(* --> NC-CAM Errors <--*)
		18944	:		FC_NcErrorMsg:='	Nc Cam Errors-	parameter:	"Table ID not allowed" The value for the table ID is not allowed, e.g. because it has already been assigned, is less than or equal to zero, or is greater than 255. 		';
		18945	:		FC_NcErrorMsg:='	Nc Cam Errors-	parameter	:	"Table type not allowed" The value for the table type is unacceptable because it is not defined. 		';
		18946	:		FC_NcErrorMsg:='	Nc Cam Errors-	parameter	:	"Number of lines in the table not allowed" The value of the number of lines in the table is not allowed, because for example, it is smaller than two at linear interpolation and smaller than four at spline interpolation. 		';
		18947	:		FC_NcErrorMsg:='	Nc Cam Errors-	parameter	:	"Number of columns in the table is not allowed" The value of the number of columns in the table is not allowed, because for example, it is less than or equal to zero (depends upon the type of table or slave). 		';
		18948	:		FC_NcErrorMsg:='	Nc Cam Errors-	parameter	:	"JogStep size (position delta) not allowed" The value for the JogStep size between two lines (position delta) is not allowed, because for example, it is less than or equal to zero. 		';
		18949	:		FC_NcErrorMsg:='	Nc Cam Errors-	parameter	:	"Period not allowed" The value for the period is not allowed, because for example, it is less than or equal to zero. 		';
		18950	:		FC_NcErrorMsg:='	Nc Cam Errors-	parameter	:	"Table is not monotonic" The value for the JogStep size is not allowed, because for example, it is less than or equal to zero.		';
		18951	:		FC_NcErrorMsg:='	Nc Cam Errors-	initialization	:	„Table sub type is not allowed” The value for the table sub type is not allowed or otherwise the table class (slave type) do not match up to the table main type.$NTable sub type: (1) equidistant linear position table, (2) equidistant cyclic position table, (3) none equidistant linear position table, (4) none equidistant cyclic position table		';
		18952	:		FC_NcErrorMsg:='	Nc Cam Errors-	initialization	:	„Table interpolation type is not allowed” The value for the table interpolation type is allowed$NTable interpolation type: (0) linear-interpolation, (1) 4-point-interpolation, (2) spline-interpolation		';
		18953	:		FC_NcErrorMsg:='	Nc Cam Errors-	initialization	:	"Incorrect table main type" The table main type is unknown or otherwise the table class (slave type) do not match up to the table main type.$NTable main type: (1) camming table, (2) characteristic table, (3) motion FUNCTION table (MF)		';
		18960	:		FC_NcErrorMsg:='	Nc Cam Errors-	initialization	:	"Table initialisation" Table has not been initialised. Although the table has been created, the rest of the initialisation has not been performed. For instance, the number of lines or columns may be less than or equal to zero.	';
		18961	:		FC_NcErrorMsg:='	Nc Cam Errors-	initialization	:	"Not enough memory" Table could not be created, since there is not enough memory.		';
		18962	:		FC_NcErrorMsg:='	Nc Cam Errors-	function	:	"Function not executed, function not available" The function has not been implemented, or cannot be executed, for the present type of table.		';
		18963	:		FC_NcErrorMsg:='	Nc Cam Errors-	function	:	"Line index not allowed" The start line index or the stop line index to be used for read or write access to the table is not allowed. $NFor instance, the line index may be greater than the total number of lines in the table.		';
		18964	:		FC_NcErrorMsg:='	Nc Cam Errors-	function	:	"Column index not allowed" The start column index or the stop column index to be used for read or write access to the table in not allowed. For instance, the column index may be greater than the total number of columns in the table.		';
		18965	:		FC_NcErrorMsg:='	Nc Cam Errors-	function	:	"Number of lines not allowed" The number of lines to be read from or written to the table is not allowed. $NThe number of lines must be an integer multiple of the number of elements in a line (n * number of columns).		';
		18966	:		FC_NcErrorMsg:='	Nc Cam Errors-	function	:	"Number of columns not allowed" The number of columns to be read from or written to the table is not allowed.$NThe number of columns must be an integer multiple of the number of elements in a column (n * number of lines).  		';
		18967	:		FC_NcErrorMsg:='	Nc Cam Errors-	function	:	"Error in scaling or in range entry" The entries in the table header are inconsistent, e.g. the validity range is empty. $NIf the error is generated during the run time it is a run time error and stops the master/slave group.		';
		18968	:		FC_NcErrorMsg:='	Nc Cam Errors-	function	:	"Multi table slave out of range" The slave master position is outside the table values for the master. The error is a run-time error, and stops the master/slave group.		';
		18969	:		FC_NcErrorMsg:='	Nc Cam Errors-	function	:	"Solo table underflow" The slave master position is outside the table values for the master. The master value of the equidistant table, to be processed linearly, lies under the first table value. $NThe error is a run-time error, and stops the master/slave group.		';
		18970	:		FC_NcErrorMsg:='	Nc Cam Errors-	function	:	"Solo table overflow" The slave master position is outside the table values for the master. The master value of the equidistant table, to be processed linearly, lies above the first table value. $NThe error is a run-time error, and stops the master/slave group.		';
		18971	:		FC_NcErrorMsg:='	Nc Cam Errors-	parameter	:	"Incorrect execution mode" The cyclic execution mode can only be "true" or "false".		';
		18972	:		FC_NcErrorMsg:='	Nc Cam Errors-	parameter	:	"Impermissible parameter" The Fifo parameter is not allowed.		';
		18973	:		FC_NcErrorMsg:='	Nc Cam Errors-	parameter	:	"Fifo is empty" The Fifo of the external generator is empty. This can signify end of track or a run time error.		';
		18974	:		FC_NcErrorMsg:='	Nc Cam Errors-	parameter	:	"Fifo is full" The Fifo of the external generator is full. It is the user‘s task to continue to attempt to fill the Fifo with the rejected values.		';
		18975	:		FC_NcErrorMsg:='	Nc Cam Errors-	parameter	:	„Point-Index of Motion Function invalid”  The point index of a Motion Function Point of a Function Table is invalid. $NFirst the point index has to be larger than zero and second it has to be numerical continuously for one column in the Montion Function Table (e.g. 1,2,3,... or 10,11,12,...).$NnRemark: The point index is not online-changeable but must be constant.		';
		18976	:		FC_NcErrorMsg:='	Nc Cam Errors-	initialization	:	„No diagonalisation of  matrix” The spline can not be calculated. The master positions are not correct.		';
		18977	:		FC_NcErrorMsg:='	Nc Cam Errors-	initialization	:	„Number of spline points to less” The number of points of a cubic spline has to be greater than two.		';
		18978	:		FC_NcErrorMsg:='	Nc Cam Errors-	initialization	:	„Fifo must not be overwritten” Fifo must not be overwritten since then the active line would be overwritten. $NIt is the task of the user to secure that the active line is not modified.		';


(* --> NC-PLC Errors <--*)

		19200	:		FC_NcErrorMsg:='NC-PLC Errors-Parameter:"Axis has been stopped" The axis has been stopped while the axis moves to target position.  The axis could be stopped with a PLC Command via ADS, with the call of AXFNC or with the TwinCAT System Manager.';
		19201	:		FC_NcErrorMsg:='NC-PLC Errors-Parameter:"Axis cannot be started" The axis cannot be started, because: the axis is in an error state, the axis is doing another job,  The axis in protected mode, the axis is not in a ready state.';
		19202	:		FC_NcErrorMsg:='NC-PLC Errors-Parameter:"Control mode not allowed" No Target Position Control and no Position Area Control.';
		19203	:		FC_NcErrorMsg:='NC-PLC Errors-Parameter:"Axis is not moving" Restart position and velocity is only allowed if axis is physically moving.';
		19204	:		FC_NcErrorMsg:='NC-PLC Errors-Parameter:"Wrong mode for RestartPosAndVelo" Wrong mode.';
		19205	:		FC_NcErrorMsg:='NC-PLC Errors-Parameter:"Command not allowed": Endless move to a non specified direction;Read/Write parameter: type mismatch';
		19206	:		FC_NcErrorMsg:='NC-PLC Errors-Parameter:"Parameter not correct"	:Wrong override: > 100% or < 0%	;Wrong gearing factor: RatioDenominator = 0	;Wrong register into process (Register communication)';
		19207	:		FC_NcErrorMsg:='NC-PLC Errors-Parameter:"Timeout axis function block":After positioning, all "MC_Move..." blocks check whether positioning was completed successfully. In the simplest case, the "AxisHasJob" flag of the NC axis is checked, which initially signifies that positioning was logically completed. Depending on the parameterisation of the NC axis,  further checks (quality criteria) are used:"Position range monitoring"	If position range monitoring is active,  the system waits for feedback from the NC.  After positioning, the axis must be within the specified positioning range window. If necessary, the position controller ensures that the axis is moved to the target position.  If the position controller is switched off (Kv=0) or weak, the target may not be reached."Target position monitoring" If target position monitoring is active, the system waits for feedback from the NC.  After positioning, the axis must be within the specified target position window for at least the specified time.  If necessary, the position controller ensures that the axis is moved to the target position.  If the position controller is switched off (Kv=0) or weak, the target may not be reached.  Floating position control may lead to the axis oscillating around the window but not remaining inside the window. If the axis is logically at the target position (logical standstill) but the parameterised position window has not been reached,  monitoring of the above-mentioned NC feedback is aborted with error 19207 (0x4B07) after a constant timeout of 6 seconds. ';
		19208	:		FC_NcErrorMsg:='NC-PLC Errors-Parameter:"Axis in protected mode" Axis is in protected mode (i.e. coupled) and cannot be moved.';
		19209	:		FC_NcErrorMsg:='NC-PLC Errors-Parameter:"Axis is not ready" Axis is not ready and cannot be moved.';
		19210	:		FC_NcErrorMsg:='NC-PLC Errors-Parameter:"Homing error" The Homing of an axis could not be started or was not successful';
		19211	:		FC_NcErrorMsg:='NC-PLC Errors-Parameter:"Invalid definition trigger input definition" The definition of the trigger signal used with the function block MC_TouchProbe is invalid.  The defined encoder ID, the trigger signal or the trigger signal edge are invalid.';
		19212	:		FC_NcErrorMsg:='NC-PLC Errors-Function:"position latch has been deactivated" The function block MC_TouchProbe encountered that a touch probe sequence has been deactivated after the block started this sequence.  The reason for instance can be an axis reset.';
		19213	:		FC_NcErrorMsg:='NC-PLC Errors-Function:"Timeout NC status feedback" A function block has successfully executed a command but the NC does not pass the expected feedback in the axis status word.';
		19214	:		FC_NcErrorMsg:='NC-PLC Errors-Function:"Supplement not installed" - The function is available as supplement product but not installed on the system.';
		19215	:		FC_NcErrorMsg:='NC-PLC Errors-Function:"Timeout Register Access" - The access to a bus terminal register timed out.';
		19216	:		FC_NcErrorMsg:='NC-PLC Errors-Function:"M-Function request missing" This error occurs if a confirmation of an M-Function is made but the request bit is not set.';
		19217	:		FC_NcErrorMsg:='NC-PLC Errors-Parameter:"Zero shift index is out of range" The index of the zero shift is invalid';
		19218	:		FC_NcErrorMsg:='NC-PLC Errors-Parameter:"R parameter index or size is invalid". This error occurs, if the R parameters are written or read and the index or size is out of range';
		19219	:		FC_NcErrorMsg:='NC-PLC Errors-Parameter:"Index for tool description is invalid"';
		19220	:		FC_NcErrorMsg:='NC-PLC Errors-Function:"Version of cyclic channel interface does not match to the requested function and function block, resp."  This error occurs, if an older TwinCAT Version is used and a new functionality from a newer TcNci.lib is called.';
		19221	:		FC_NcErrorMsg:='NC-PLC Errors-Function:"Channel is not ready for requested function". The requested function can not be executed due to a wrong state of the channel.  This error occurs for instance, if retrace is requested and the axes are not stopped with ItpEStop before.';
		19222	:		FC_NcErrorMsg:='NC-PLC Errors-Function:"Requested function is not turned on". The requested function requires an explicit activation before it can be executed.';
		19232	:		FC_NcErrorMsg:='NC-PLC Errors-Parameter:"Cannot append all axes". This error occurs, if you want to append an auxiliary axes to an interpolation group and the function fails.  Probably a prior assignment of an auxiliary axes was skipped.';
		19248	:		FC_NcErrorMsg:='NC-PLC Errors-Parameter:"Pointer invalid". The pointer to a data structure is invalid, e.g. NULL.:data structure MC_CAM_REF is possibly not initialized';
		19249	:		FC_NcErrorMsg:='NC-PLC Errors-Parameter:"Size of memory invalid". The size parameter is invalid:The value of the size parameter is 0 or less than the size of one element of the addressed data structure. The value of the size parameter is less than the requested amount of data. The value of the size parameter does not match other parameters as number of points, number of rows or number of columns.';
		19250	:		FC_NcErrorMsg:='NC-PLC Errors-Parameter:"Invalid cam table ID". The cam table ID is out of the range from 1 to 255.';
		19251	:		FC_NcErrorMsg:='NC-PLC Errors-Parameter:"Invalid point ID". The point ID of a motion function point is lower than 1.';
		19252	:		FC_NcErrorMsg:='NC-PLC Errors-Parameter:"Invalid number of points ". The number of points to read or write is less than 1.';
		19253	:		FC_NcErrorMsg:='NC-PLC Errors-Parameter:"Invalid MC table type". The type of a cam table does not match the MC_TableType definition.';
		19254	:		FC_NcErrorMsg:='NC-PLC Errors-Parameter:"Invalid number of rows". The number of rows of a cam table is less than 1.';
		19255	:		FC_NcErrorMsg:='NC-PLC Errors-Parameter:"Invalid number of columns". The number of columns of a cam table is invalid. The number of columns of a motion function is not equal to 1 ;The number of columns of a standard cam table is not equal to 2 The number of columns does not match other parameters (ValueSelectMask)';
		19256	:		FC_NcErrorMsg:='NC-PLC Errors-Parameter:"Invalid Increment". The increment for an interpolation is invalid, e.g. <= 0.';
		19264	:		FC_NcErrorMsg:='NC-PLC Errors-Monitoring:"Unsupported Terminal Type". The terminal in use is not supported by this function block.';
		19265	:		FC_NcErrorMsg:='NC-PLC Errors-Monitoring:"Register Read/Write Error". This error implies to be a validation error.';
		19266	:		FC_NcErrorMsg:='NC-PLC Errors-Monitoring:"Axis is Enabled". Axis is enabled and is not supposed to be enabled for this operation';
		19267	:		FC_NcErrorMsg:='NC-PLC Errors-Parameter:"Size of compensation table wrong". The stated table size in bytes is not conform with the real size.';
		19268	:		FC_NcErrorMsg:='NC-PLC Errors-Parameter:The minimum/ maximum position of the compenstation table is not conform to the position in the table description (ST_CompensationDesc)';
		19269	:		FC_NcErrorMsg:='NC-PLC Errors-Parameter:"Not implemented". The requested function is not implemented in this combination.';
		19296	:		FC_NcErrorMsg:='NC-PLC Errors-Monitoring:"Motion command not be activated". A motion command has been started and has been buffered and confirmed by the NC. Nevertheless the command did not become active.';
		19297	:		FC_NcErrorMsg:='NC-PLC Errors-Monitoring:"Motion command could not be monitored by the PLC". A motion command has been started and has been buffered and confirmed by the NC.  The PLC has not been able to monitor the execution of this command and the execution status is unclear since the NC is already executing a more recent command.  This error may com up with very short buffered motion commands which are executed during one PLC cycle.';
		19298	:		FC_NcErrorMsg:='NC-PLC Errors-Monitoring:"Buffered command finished with error". A buffered command finished with an error. The error number is not available because a new command is already in execution.';
		19299	:		FC_NcErrorMsg:='NC-PLC Errors-Monitoring:"Buffered command finished without state feedback". A buffered command finished without success or error feedback.';
		19300	:		FC_NcErrorMsg:='NC-PLC Errors-Monitoring:" "BufferMode" not supported". The "BufferMode" is not supported by the command.';
		19301	:		FC_NcErrorMsg:='NC-PLC Errors-Monitoring:"Command number is zero". The system administrated command number for buffered commands is zero.';
		19313	:		FC_NcErrorMsg:='NC-PLC Errors-Parameter:"Invalid NCI Entry Type". FB_NciFeedTablePreparation is called with an unknown nEntryType';
		19314	:		FC_NcErrorMsg:='NC-PLC Errors-Function:"NciFeedTable full". The table is full filled and therefore this entry is not accepted. To do:Transfer the context of the table with FB_NciFeedTable to the NC-Kernel.  If this succeeded bFeedingDone becomes TRUE and the context of the table has to be reset with bResetTable (FB_NciFeedTablePreparation).  Now the table can be refilled with new entries.';
		19315	:		FC_NcErrorMsg:='NC-PLC Errors-Function:internal error';
		19316	:		FC_NcErrorMsg:='NC-PLC Errors-Parameter:$NST_NciTangentialFollowingDesc: tangential axis is not an auxiliary axis"  The entry ST_NciTangentialFollowingDesc contains an tangential axis that is no auxiliary axis.';
		19317	:		FC_NcErrorMsg:='NC-PLC Errors-Parameter:$NST_NciTangentialFollowingDesc: nPathAxis1 and nPathAxis2, resp. are no path axes. So it is not possible to determine the plane.';
		19318	:		FC_NcErrorMsg:='NC-PLC Errors-Parameter:$NST_NciTangentialFollwoingDesc: nPathAxis1 and nPathAxis2 are equal. So it is not possible to determine the plane.';
		19319	:		FC_NcErrorMsg:='NC-PLC Errors-Parameter:$NST_NciGeoCirclePlane: circle is programmed in a wrong manner.';
		19320	:		FC_NcErrorMsg:='NC-PLC Errors-Function:$NInternal error in calculation of the tangential following';
		19321	:		FC_NcErrorMsg:='NC-PLC Errors-Monitoring:$NTangential following: With ST_NciTangentialFollowingDesc the monitoring of the deviation angle (E_TfErrorOnCrirical1)  is activated and with the actual segment the deviation angle is too big.';
		19322	:		FC_NcErrorMsg:='NC-PLC Errors-Function:$Nnot implemented';
		19323	:		FC_NcErrorMsg:='NC-PLC Errors-Parameter:$NTangential Following: The radius of the actual circle segment is too small';
		19324	:		FC_NcErrorMsg:='NC-PLC Errors-Parameter:$NFB_NciFeedTablePreparation: pEntry is NULL';
		19325	:		FC_NcErrorMsg:='NC-PLC Errors-Parameter:$NFB_NciFeedTablePreparation: The specified nEntryType does not match the the structure type';
		19326	:		FC_NcErrorMsg:='NC-PLC Errors-Parameter:$NST_NciMFuncFast and ST_NciMFuncHsk: The requested m-function is not in between 0..159';
		19327	:		FC_NcErrorMsg:='NC-PLC Errors-Parameter:$NST_NciDynOvr: The requested value for the dynamic override is not in between 0.01 and 1.0';
		19328	:		FC_NcErrorMsg:='NC-PLC Errors-Parameter:$NST_NciVertexSmoothing: invalid parameter. This error occurs with a negative vertex radius or an unknown vertex smoothing type.';
		19329	:		FC_NcErrorMsg:='NC-PLC Errors-Parameter:$NFB_NciFeedTablePrepartion: The requested velocity is not in a valid range';
		19330	:		FC_NcErrorMsg:='NC-PLC Errors-Parameter:$NST_Nci*: invalid parameter';



		33056	:	FC_NcErrorMsg:='NC3_Environment_Invalid configuration for Object (e.g. in System Manager)';
		33057	:	FC_NcErrorMsg:='NC3_Environment_Invalid environment FOR Object (e.g. TcCom-Object Hierarchy OR missing/faulty Objects)';
		33058	:	FC_NcErrorMsg:='NC3_Environment_Incompatible Driver OR Object';
		33084	:	FC_NcErrorMsg:='NC3_Parameter_BufferMode is invalid';
		33085	:	FC_NcErrorMsg:='NC3_FunctionBlock_Only one active Instance OF FUNCTION Block per Group is allowed';
		33086	:	FC_NcErrorMsg:='NC3_State_Command is NOT allowed in current group state';
		33087	:	FC_NcErrorMsg:='NC3_FunctionBlock_Slave cannot synchronize.The slave cannot reach the SlaveSyncPosition BY the TIME the master has reached the MasterSyncPos';
		33088	:	FC_NcErrorMsg:='NC3_Parameter_Invalid value FOR one OR more OF the dynamic parameters (A, D, J)';
		33089	:	FC_NcErrorMsg:='NC3_Parameter_IdentInGroup is invalid';
		33090	:	FC_NcErrorMsg:='NC3_Parameter_The number OF axes in the group is incompatible with the axes convention';
		33091	:	FC_NcErrorMsg:='NC3_Communication_FUNCTION Block OR respective Command is NOT supported BY Target';
		33093	:	FC_NcErrorMsg:='NC3_FunctionBlock_Mapping OF Cyclic INTERFACE between Nc AND Plc missing (e.g. AXIS_REF, AXES_GROUP_REF, ...)';
		33094	:	FC_NcErrorMsg:='NC3_FunctionBlock_Invalid Velocity ValueThe velocity was NOT set OR the entered value is invalid';
		33096	:	FC_NcErrorMsg:='NC3_FunctionBlock_Invalid Input Value';
		33097	:	FC_NcErrorMsg:='NC3_FunctionBlock_Invalid OR Incomplete Input ARRAY';
		33098	:	FC_NcErrorMsg:='NC3_Parameter_Unsupported Dynamics FOR selected Group Kernel';
			
		
		ELSE
			IF 36844<error AND error< 36857 THEN
				FC_NcErrorMsg:='NC3_Internal_Unexpected INTERNAL Error';
			ELSE		
				FC_NcErrorMsg:='Msg Unknown';
			END_IF	
END_CASE

END_FUNCTION

// ---- POUs/Lib/Motion/CreateNCErrMsgDetails.TcPOU
FUNCTION CreateNCErrMsgDetails : enumMotorEvents
VAR_INPUT
	Error: UDINT;
END_VAR
VAR
END_VAR

CASE Error OF
		0		: 		
(* --> General NC Errors <--*)
			CreateNCErrMsgDetails := enumMotorEvents.NoEvents;
		16384,16385,16386,16400,16401,16402,16403,16404,16405,16406	:	
			CreateNCErrMsgDetails := enumMotorEvents.MotorGeneralError;
		16416,16417,16418,16419,16420,16421	:
			CreateNCErrMsgDetails := enumMotorEvents.MotorFeedBackErr;
		16432,16433,16448:	
			CreateNCErrMsgDetails := enumMotorEvents.MotorGeneralError;
		16464	,	16465	,16466	:	
			CreateNCErrMsgDetails := enumMotorEvents.MotorFeedBackErr;
		16480,16481	,16482	,16483	,16496	,16497	:		
            CreateNCErrMsgDetails := enumMotorEvents.MotorGeneralError;      
                        
(* --> Channel Errors <-*)
		16641	,	
		16642	,	
		16643	,	
		16644	,	
		16645	,	
		16646	,	
		16647	,	
		16648	,	
		16649	,	
		16650	,	
		16656	,	
		16657	,	
		16658	,	
		16659	,	
		16660	,	
		16661	,	
		16662	,	
		16663	,	
		16672	,
		16673	,	
		16674	,	
		16688	,	
		16689	,	
		16690	,	
		16691	,	
		16704	,	
		16705	,	
		16706	,	
		16707	,	
		16708	,	
		16709	,	
		16720	,	
		16721	,	
		16722	,	
		16723	,	
		16724	,	
		16725	,
		16726	,	
		16727	,	
		16728	,	
		16729	,	
		16730	,	
		16731	,	
		16732	,	
		16733	,	
		16734	,
		16735	,
		16736	,	
		16737	,	
		16738	,	
		16752	,	
		16753	,	
		16754	:	
 			CreateNCErrMsgDetails := enumMotorEvents.MotorGeneralError; 
(* --> Group Errors <--*)

		16896	,	
		16897	,	
		16898	,	
		16899	,	
		16900	,	
		16901	,	
		16902	,	
		16903	,	
		16904	,	
		16905	,	
		16906	,	
		16907	,	
		16908	,	
		16909	,	
		16910	,	
		16911	,	
		16912	,	
		16913	,	
		16914	,	
		16915	,	
		16916	,	
		16917	,	
		16918	,	
		16919	,	
		16920	,	
		16921	,	
		16922	,	
		16923	,	
		16924	,	
		16925	,	
		16926	,	
		16927	,	
		16928	,	
		16929	,	
		16930	:
				CreateNCErrMsgDetails := enumMotorEvents.PLCIllegalParam; 
		16931	:
				CreateNCErrMsgDetails := enumMotorEvents.DriveNotEnabled; 	
		16932	:
				CreateNCErrMsgDetails := enumMotorEvents.MotorGeneralError ;
		16933	:
				CreateNCErrMsgDetails := enumMotorEvents.DriveNotReady ;	
		16934	,	
		16935	:	;
				
		16936	,	
		16937	:	;
				CreateNCErrMsgDetails := enumMotorEvents.MotorGeneralError;	
		16938	:
				CreateNCErrMsgDetails := enumMotorEvents.DriveNotEnabled; 		
		16939	,	
		16940	,	
		16941	,	
		16942	,	
		16943	,	
		16944	,	
		16945	,	
		16946	,	
		16947	,	
		16948	:	;
		16949	,	
		16950	,	
		16951	,	
		16952	,	
		16953	,	
		16954	,	
		16955	,	
		16956	,	
		16957	:	;
		16958	,	
		16959	,	
		16960	,	
		16961	,	
		16962	,	
		16963	,	
		16964	,	
		16965	,	
		16966	:	;
		16967	,	
		16968	,	
		16969	,	
		16970	,	
		16971	,	
		16972	,	
		16973	,	
		16974	,	
		16975	:	;
		16976	,	
		16977	,	
		16978	,	
		16979	:
				CreateNCErrMsgDetails := enumMotorEvents.MotorGeneralError;		
		16980	:
				CreateNCErrMsgDetails := enumMotorEvents.MotorFeedBackErr;			
		16981	,	
		16982	,	
		16983	,	
		16984	:	;
		16985	,	
		16986	,	
		16987	,	
		16988	,	
		16989	,	
		16990	,	
		16991	:
		 		CreateNCErrMsgDetails := enumMotorEvents.MotorGeneralError;	
		16992	:	
				CreateNCErrMsgDetails := enumMotorEvents.DriveNotEnabled ;
		16993	,	
		16994	,	
		16995	,	
		16996	,	
		16997	,	
		16998	,	
		16999	,	
		17000	,	
		17001	,	
		17002	,	
		17003	,	
		17004	,	
		17005	,	
		17006	,	
		17007	,	
		17008	,	
		17009	,	
		17010	,	
		17011	,	
		17012	,	
		17014	,	
		17015	,	
		17017	,	
		17018	,	
		17019	,	
		17020	,	
		17021	,	
		17022	,	
		17023	,	
		17024	,	
		17025	,	
		17026	,	
		17027	,	
		17028	,	
		17029	,	
		17030	,	
		17031	,	
		17032	,	
		17033	,	
		17034	,	
		17035	,	
		17036	,	
		17037	,
		17038	,
		17039	,
		17040	,
		17041	,
		17042	,
		17043	,
		17044	,
		17045	,
		17046	,
		17047	,
		17052	,
		17053	,
		17054	,
		17056	,	
		17057	,	
		17058	,	
		17059	,	
		17060	,	
		17061	,	
		17062	,	
		17063	,	
		17064	,	
		17065	,	
		17066	,	
		17067	,	
		17068	,	
		17069	,	
		17070	,	
		17071	,	
		17072	,	
		17073	,	
		17074	,	
		17075	,	
		17076	,	
		17077	,	
		17078	,	
		17079	,	
		17080	,	
		17082	,	
		17083	,	
		17084	,	
		17085	,	
		17086	,		
		17087	,		
		17088	,		
		17089	,		
		17090	,		
		17091	,		
		17092	,		
		17093	,		
		17094	,		
		17095	,		
		17096	,		
		17097	,		
		17098	,		
		17099	,		
		17100	,		
		17101	,		
		17102	,		
		17103	,		
		17104	,		
		17105	,		
		17106	,		
		17107	,		
		17108	,		
		17109	,		
		17110	,		
		17111	,		
		17112	,		
		17114	,		
		17115	,		
		17116	,		
		17117	,		
		17118	,		
		17119	,		
		17120	,		
		17121	,		
		17122	,		
		17123	,		
		17124	,		
		17125	,		
		17127	,		
		17128	,		
		17129	,		
		17130	,		
		17131	,		
		17132	,		
		17133	,		
		17134	,		
		17135	,		
		17136	,		
		17137	,		
		17138	,		
		17139	,		
		17140	,		
		17142	,		
		17151	:		
               CreateNCErrMsgDetails := enumMotorEvents.MotorGeneralError;	         

(* --> Axis Errors <--*)

		17152	,		
		17153	,		
		17158	,		
		17159	,		
		17160	,		
		17161	,		
		17162	,		
		17163	,		
		17164	,		
		17165	,		
		17166	,		
		17167	,		
		17168	,		
		17170	,		
		17171	,		
		17172	,		
		17173	,		
		17174	,		
		17175	,		
		17176	,		
		17177	,		
		17178	,		
		17179	,		
		17180	,		
		17181	,		
		17182	,		
		17183	,		
		17184	,		
		17185	,		
		17186	,		
		17187	,		
		17188	,		
		17189	,		
		17190	,		
		17191	,		
		17192	,		
		17193	,		
		17194	,		
		17195	,		
		17196	,		
		17197	,		
		17198	,		
		17199	,		
		17200	,		
		17201	,		
		17202	,		
		17203	,		
		17204	,		
		17210	,		
		17211	:	
				CreateNCErrMsgDetails := enumMotorEvents.MotorGeneralError;		
		17216	:		
				CreateNCErrMsgDetails := enumMotorEvents.DriveNotReady ;
		17217	,		
		17218	,		
		17219	,		
		17220	,		
		17221	,		
		17222	,		
		17223	,		
		17224	:
			CreateNCErrMsgDetails := enumMotorEvents.MotorGeneralError;				
		17238	,		
		17239	,		
		17240	:
			CreateNCErrMsgDetails := enumMotorEvents.DriveNotEnabled;
		17241	,		
		17242	,		
		17243	,		
		17244	:
				CreateNCErrMsgDetails := enumMotorEvents.MotorGeneralError;		
		17245	:
				CreateNCErrMsgDetails := enumMotorEvents.MotorPositionError;		
		17246	,		
		17249	,		
		17250	,		
		17251	,		
		17312	:		
	             CreateNCErrMsgDetails := enumMotorEvents.MotorGeneralError;
                        
(* --> Encoder Errors <--*)           
		17408	,		
		17409	,		
		17410	,		
		17411	,		
		17412	,		
		17413	,		
		17414	,		
		17415	,		
		17416	,		
		17417	,		
		17418	,		
		17419	,		
		17420	,		
		17421	,		
		17422	,		
		17423	,		
		17424	,		
		17425	,		
		17426	,		
		17427	,		
		17428	,		
		17429	,		
		17430	,		
		17431	,		
		17432	,		
		17433	,		
		17434	,		
		17435	,		
		17436	,		
		17440	,		
		17441	,		
		17442	,		
		17443	,		
		17444	,		
		17445	,		
		17446	,		
		17456	,		
		17457	,		
		17458	,		
		17459	,		
		17460	,		
		17461	:		
		        CreateNCErrMsgDetails := enumMotorEvents.MotorGeneralError;
		17472	:
				CreateNCErrMsgDetails := enumMotorEvents.DriveNotReady;		
		17473	,	
		17474	,		
		17475	:
  				CreateNCErrMsgDetails := enumMotorEvents.MotorGeneralError;		
		17488	,  				
		17489	:
				CreateNCErrMsgDetails := enumMotorEvents.MotorFeedBackErr;				
		17504	,		
		17505	,		
		17506	,		
		17507	:
				CreateNCErrMsgDetails := enumMotorEvents.MotorGeneralError;				
		17508	,		
		17509	:
				CreateNCErrMsgDetails := enumMotorEvents.MotorFeedBackErr;
			
		17510   :
				CreateNCErrMsgDetails := enumMotorEvents.DriveComError;
	 
		17520	,	
		17570	,	
		17571	:
			CreateNCErrMsgDetails := enumMotorEvents.MotorGeneralError;	

(* --> Controller Errors <--*)
		17664	,
		17665	, 
		17666	,
		17667	,
		17668	,
		17669	,
		17670	,
		17671	,
		17672	,
		17673	,
		17680	,
		17681	,
		17682	,
		17683	,
		17684	,
		17685	,
		17686	,
		17687	,
		17688	,
		17689	,
		17690	,
		17691	,
		17692	,
		17693	,
		17696	,
		17697	,
		17698	,
		17699	,
		17700	:
			CreateNCErrMsgDetails := enumMotorEvents.MotorGeneralError;	
		17728	:
			CreateNCErrMsgDetails := enumMotorEvents.DriveNotReady;
		17729	,	
		17730	:
			CreateNCErrMsgDetails := enumMotorEvents.MotorGeneralError;		
		17744	:
			CreateNCErrMsgDetails := enumMotorEvents.MotorPositionError;
		17745	:
			CreateNCErrMsgDetails := enumMotorEvents.MotorSpeedError;
		17824	,	
		17825	,	
		17826	,	
		17827	,	
		17828	:	
			CreateNCErrMsgDetails := enumMotorEvents.MotorGeneralError;	

(* --> Drive Errors <--*)

		17920	,
		17921	,
		17922	,
		17923	,
		17924	,
		17925	,
		17926	,
		17927	,
		17928	,
		17929	,
		17930	, 
		17931	,
		17932	,
		17933	,
		17935	,
		17936	,
		17937	,	
		17938	,
		17939	,
		17940	,
		17941	,
		17942	,
		17943	,
		17952	,
		17953	,
		17954	,
		17955	,
		17956	,
		17959	:
			CreateNCErrMsgDetails := enumMotorEvents.MotorGeneralError;	

		17968	:
			CreateNCErrMsgDetails := enumMotorEvents.MotorOverTemp;	
		17969	,
		17970	,
		17971	:
			CreateNCErrMsgDetails := enumMotorEvents.MotorSupplyError;
		17972	,
		17973	:
			CreateNCErrMsgDetails := enumMotorEvents.MotorOverCurrent;
		17974	:
			CreateNCErrMsgDetails := enumMotorEvents.MotorStalled;
		17984	:
			CreateNCErrMsgDetails := enumMotorEvents.DriveNotReady;
		17985	,
		17986	,
		17987	:
			CreateNCErrMsgDetails := enumMotorEvents.MotorGeneralError;	
		18000	:
			CreateNCErrMsgDetails := enumMotorEvents.DriveNotReady;	
		18001	:
			CreateNCErrMsgDetails := enumMotorEvents.DriveComError;
		18002	:
			CreateNCErrMsgDetails := enumMotorEvents.MotorGeneralError;	
		18005	:
			CreateNCErrMsgDetails := enumMotorEvents.DriveComError;

(* --> NC-CAM Errors <--*)
		18944	, 
		18945	, 
		18946	, 
		18947	, 
		18948	, 
		18949	, 
		18950	, 
		18951	, 
		18952	, 
		18953	, 
		18960	, 
		18961	, 	
		18962	, 	
		18963	, 
		18964	, 
		18965	, 
		18966	,	
		18967	, 
		18968	, 	
		18969	, 
		18970	, 
		18971	, 	
		18972	,	
		18973	,	
		18974	,	
		18975	,
		18976	,	
		18977	,	
		18978	,	
		18979   : 
			CreateNCErrMsgDetails := enumMotorEvents.MotorGeneralError;
(* --> NC-PLC Errors <--*)

		19200	,	
		19201	,	
		19202	,	
		19203	,	
		19204	,	
		19205	,	
		19206	,	
		19207	,
		19208	,	
		19209	,	
		19210	,	
		19211	,	
		19212	,	
		19213	,	
		19214	,	
		19215	,	
		19216	,	
		19217	,
		19218	,
		19219	,
		19220	,
		19221	,
		19222	,
		19232	,
		19248	:	;
		19249	,
		19250	,
		19251	,
		19252	,
		19253	,
		19254	,
		19255	,
		19256	,
		19264	,
		19265	,
		19266	,
		19267	,
		19268	,
		19269	,
		19296	,
		19297	,
		19298	,
		19299	,
		19300	,
		19301	,
		19313	,
		19314	,
		19315	,
		19316	,
		19317	,
		19318	,
		19319	,
		19320	,
		19321	,
		19322	,
		19323	,
		19324	,
		19325	,
		19326	,
		19327	,
		19328	,
		19329	,
		19330	,
		19344   ,
		19345   ,
		19346   ,
		19347   ,
		19348   ,
		19349   ,
		19350   ,
		19351   ,
		19352   ,
		19360   ,
		19361   ,
		19376   ,
		19377   ,
		19378   ,
		19379   ,
		19380   ,
		19381   :
                
            	CreateNCErrMsgDetails := enumMotorEvents.MotorGeneralError;    
		        
                
                
		33056	,
		33057	,
		33058	,
		33084	,
		33085	,
		33086	,
		33087	,
		33088	,
		33089	,
		33090	,
		33091	,
		33093	,
		33094	,
		33096	,
		33097	,
		33098	:	
				CreateNCErrMsgDetails := enumMotorEvents.MotorGeneralError;
		
		ELSE
			IF 36844<error AND error< 36857 THEN
			//
			ELSE		
				//
				CreateNCErrMsgDetails := enumMotorEvents.MotorGeneralError;
			END_IF	
END_CASE

END_FUNCTION

// ---- POUs/Lib/Motion/MultiAxis_FB.TcPOU
FUNCTION_BLOCK PUBLIC MultiAxis_FB
VAR_INPUT
	
	BasicAxisCtrlPtr 	: POINTER TO Basic_axis_typ ;
	MultiAxisCtrlPtr 	: POINTER TO MultiAxis_typ ;
	
END_VAR
VAR_IN_OUT
	MasterRef	:	AXIS_REF;
    MasterRef2 	: 	AXIS_REF;
    MasterRef3 	: 	AXIS_REF;
    MasterRef4 	: 	AXIS_REF;
	AxisRef		: 	AXIS_REF;
END_VAR
VAR_OUTPUT
END_VAR
	
VAR
	LogMsgInit		: BOOL;
	LogMsg_0 		: LogMsg ;
	DecoupleTriger	: Trigger ;
	Decouple		: bool ;
	fbMC_CamTableSelect	: MC_CamTableSelect;
	fbMC_CamIn			: MC_CamIn;
	fbMC_CamOut			: MC_CamOut;
	fbMC_GearInDyn		: MC_GearInDyn;
	fbMC_GearInPos		: MC_GearInPos;
	fbMC_GearOut		: MC_GearOut ;
	fbMC_GearInMultiMaster : MC_GearInMultiMaster ;
	
	ErrorTrig : Trigger ;
	AxisStep : eMultiAxisState ;
	tempTrig : Trigger ;
	
	
	
	tmp_ErrorEntry			: Eh_ErrorEntry_typ;
	
END_VAR

IF NOT LogMsgInit THEN 
	LogMsg_0.logData.category:=	BasicAxisCtrlPtr^.Input.Parameter.ThreadName;     
	LogMsg_0.Enable:= 	TRUE; 	
END_IF

LogMsg_0.ptrGlobalArray:= 	ADR(LogGlobalArray);
LogMsg_0.ptrEncoderAngle:= 	ADR(BasicAxisCtrlPtr^.Input.Parameter.PosForLog);

IF BasicAxisCtrlPtr^.Output.Status.FAULT THEN
	

	AxisStep := MultiAxis_STATE_ERROR;
		
END_IF

//in case of Stop go to CAM_STATE_WAIT
IF (BasicAxisCtrlPtr^.Input.Command.Stop = TRUE) OR (BasicAxisCtrlPtr^.Input.Command.Halt = TRUE) THEN
	AxisStep := MultiAxis_STATE_WAIT;
END_IF

CASE AxisStep OF
		
	(******************** WAIT *************************)
	MultiAxis_STATE_WAIT:  (* STATE: Wait *)
		
		IF BasicAxisCtrlPtr^.Output.Status.ReadyForCmd THEN
			Disable_All_FB(FALSE);
			AxisStep := MultiAxis_STATE_ENTER_READY ;
		END_IF
		
	MultiAxis_STATE_ENTER_READY:
			IF Disable_All_FB(TRUE) THEN
				AxisStep := MultiAxis_STATE_READY ;
			END_IF	

	(******************** READY *************************)
	MultiAxis_STATE_READY:
	
		IF MultiAxisCtrlPtr^.Input.Command.CamTableSelect.Start THEN
			
			MultiAxisCtrlPtr^.Input.Command.CamTableSelect.Start := FALSE ;
			MultiAxisCtrlPtr^.Output.Status.CamTableSelect.Done := FALSE ;
			AxisStep := MultiAxis_STATE_CAM_SELECT ;
			
		ELSIF MultiAxisCtrlPtr^.Input.Command.CamIn.StartSlave THEN
			
			MultiAxisCtrlPtr^.Input.Command.CamIn.StartSlave := FALSE ;
			fbMC_CamIn.Execute := FALSE;	
			AxisStep := MultiAxis_STATE_CAM_START ;
			
		ELSIF MultiAxisCtrlPtr^.Input.Command.CamIn.DisengageSlave THEN
			
			MultiAxisCtrlPtr^.Input.Command.CamIn.DisengageSlave := FALSE ;
			MultiAxisCtrlPtr^.Output.Status.CamOut.Done := FALSE ;
			fbMC_CamOut.Execute := FALSE ;
			AxisStep := MultiAxis_STATE_CAM_STOP ;
			
		ELSIF MultiAxisCtrlPtr^.Input.Command.GearInPos.StartSlave  THEN
			MultiAxisCtrlPtr^.Input.Command.GearInPos.StartSlave := FALSE ;
			MultiAxisCtrlPtr^.Output.Status.GearInPos.InSync := FALSE ;
			MultiAxisCtrlPtr^.Output.Status.GearOut.Done 	:= FALSE ;
			AxisStep := MultiAxis_STATE_GEAR_IN_POS ;
			
		ELSIF MultiAxisCtrlPtr^.Input.Command.GearInDyn.StartSlave THEN
			MultiAxisCtrlPtr^.Input.Command.GearInDyn.StartSlave := FALSE ;
			MultiAxisCtrlPtr^.Output.Status.GearInDyn.InGear := FALSE ;
			MultiAxisCtrlPtr^.Output.Status.GearOut.Done 	:= FALSE ;
			AxisStep := MultiAxis_STATE_GEAR_IN_DYN ;
			
		ELSIF MultiAxisCtrlPtr^.Input.Command.GearInDyn.DisengageSlave THEN
			MultiAxisCtrlPtr^.Input.Command.GearInDyn.DisengageSlave := FALSE ;
			MultiAxisCtrlPtr^.Output.Status.GearInDyn.InGear := FALSE ;
			MultiAxisCtrlPtr^.Output.Status.GearOut.Done 	:= FALSE ;
			MultiAxisCtrlPtr^.Output.Status.GearInMultiMaster.InGear := FALSE ;
			AxisStep := MultiAxis_STATE_GEAR_OUT ;
			
		ELSIF MultiAxisCtrlPtr^.Input.Command.GearInMultiMaster.StartSlave THEN
			MultiAxisCtrlPtr^.Input.Command.GearInMultiMaster.StartSlave := FALSE ;
			MultiAxisCtrlPtr^.Output.Status.GearInMultiMaster.InGear := FALSE ;
			MultiAxisCtrlPtr^.Output.Status.GearOut.Done 	:= FALSE ;
			AxisStep := MultiAxis_STATE_GEAR_IN_MULTI_MASTER;
			
		ELSIF MultiAxisCtrlPtr^.Input.Command.GearInMultiMaster.DisengageSlave THEN
			MultiAxisCtrlPtr^.Input.Command.GearInMultiMaster.DisengageSlave := FALSE ;
			MultiAxisCtrlPtr^.Output.Status.GearInDyn.InGear := FALSE ;
			MultiAxisCtrlPtr^.Output.Status.GearOut.Done 	:= FALSE ;
			MultiAxisCtrlPtr^.Output.Status.GearInMultiMaster.InGear := FALSE ;
			AxisStep := MultiAxis_STATE_GEAR_OUT ;
		END_IF
	
	(******************** CamTableSelect *************************)	
	MultiAxis_STATE_CAM_SELECT:

		IF THIS^.CamTableSelect()THEN
			AxisStep := MultiAxis_STATE_READY;
		END_IF
		
	(******************** START CAM MOVEMENT **********************)	
	MultiAxis_STATE_CAM_START:
	
		fbMC_CamIn.MasterOffset 	:= MultiAxisCtrlPtr^.Input.Parameter.CamIn.MasterOffset;
		fbMC_CamIn.SlaveOffset 		:= MultiAxisCtrlPtr^.Input.Parameter.CamIn.SlaveOffset; 
		fbMC_CamIn.MasterScaling	:= MultiAxisCtrlPtr^.Input.Parameter.CamIn.MasterScaling;
		fbMC_CamIn.SlaveScaling 	:= MultiAxisCtrlPtr^.Input.Parameter.CamIn.SlaveScaling;
		fbMC_CamIn.StartMode 		:= MultiAxisCtrlPtr^.Input.Parameter.CamIn.StartMode;
		fbMC_CamIn.CamTableID 		:= MultiAxisCtrlPtr^.Input.Parameter.CamIn.CamTableID;
		fbMC_CamIn.BufferMode 		:= MultiAxisCtrlPtr^.Input.Parameter.CamIn.BufferMode;
		fbMC_CamIn.Options 			:= MultiAxisCtrlPtr^.Input.Parameter.CamIn.Options; 
		
		fbMC_CamIn.Execute := TRUE;
		AxisStep := MultiAxis_STATE_READY;
		
	(******************** STOP CAM MOVEMENT **********************)
	MultiAxis_STATE_CAM_STOP: (* STATE: Stop electronic gear coupling *)
		
		IF THIS^.CamOut()THEN
			fbMC_CamIn.Execute := FALSE;
			AxisStep := MultiAxis_STATE_READY;
		END_IF	
			
	(******************** GEAR IN DYNAMIC **********************)	
	MultiAxis_STATE_GEAR_IN_DYN:
	
	
		IF (MultiAxisCtrlPtr^.Input.Command.GearInDyn.DisengageSlave)			 
				AND NOT THIS^.GearInDyn() THEN
			AxisStep := MultiAxis_STATE_GEAR_OUT;
		END_IF
				
	(******************** GEAR IN POSITION **********************)
	MultiAxis_STATE_GEAR_IN_POS:
	
		IF MultiAxisCtrlPtr^.Input.Command.GearInPos.DisengageSlave AND NOT THIS^.GearInPos() THEN
			AxisStep := MultiAxis_STATE_GEAR_OUT;
		END_IF
		
		//THIS^.GearInPos();

	(******************** GEAR IN MultiMaster **********************)
	MultiAxis_STATE_GEAR_IN_MULTI_MASTER:
(*	
		IF ((MultiAxisCtrlPtr^.Input.Command.GearInMultiMaster.DisengageSlave) OR (BasicAxisCtrlPtr^.Input.Command.Power = FALSE))  
			AND NOT THIS^.GearInMultiMaster() THEN
				AxisStep := MultiAxis_STATE_GEAR_OUT;
		END_IF
*)

		IF NOT THIS^.GearInMultiMaster() THEN
				AxisStep := MultiAxis_STATE_GEAR_OUT;
		END_IF
			
	(******************** GEAR OUT **********************)	
	MultiAxis_STATE_GEAR_OUT:
		
		IF THIS^.GearOut()THEN
			MultiAxisCtrlPtr^.Output.Status.GearInPos.InSync := FALSE ;
			MultiAxisCtrlPtr^.Output.Status.GearInDyn.InGear := FALSE ;
			MultiAxisCtrlPtr^.Output.Status.GearInMultiMaster.InGear := FALSE ;
			AxisStep := MultiAxis_STATE_READY;
		END_IF
		
	(******************** Error **********************)	
	MultiAxis_STATE_ERROR:	
		
			THIS^.ResetAll_MC_FB();	
		
			IF BasicAxisCtrlPtr^.Output.Status.FAULT THEN						
				AxisStep := MultiAxis_STATE_ERROR;
			ELSE
				MultiAxisCtrlPtr^.Output.Error.ErrorID := 0 ;
				AxisStep := MultiAxis_STATE_WAIT;
			END_IF			
	
	
END_CASE 


IF DecoupleTriger.EDGEPOS(BasicAxisCtrlPtr^.Output.Status.AxisStatus.Error)THEN
	Decouple := TRUE ;
END_IF
IF Decouple THEN	
	IF THIS^.GearOut() THEN
		Decouple := FALSE ;
	END_IF
END_IF

(********************** MC_CAMIN FB Call *************************)
	
THIS^.CamIn();
	
//=====================================================================================================================\\

//IF MultiAxisCtrlPtr^.Output.Error.ErrorID <> 0 THEN
//	BasicAxisCtrlPtr^.Output.Error.ErrorID := MultiAxisCtrlPtr^.Output.Error.ErrorID ;
//	MultiAxisCtrlPtr^.Output.Error.ErrorID := 0;
//END_IF

//fnLogTransfer FUNCTION call
fnLogTransfer(ADR(LogMsg_0));

METHOD AddNCError : BOOL
VAR_INPUT
	ErrorId			: UDINT;
	ErrorPrefix     : STRING[100];
END_VAR

	tmp_ErrorEntry.ErrorId		:= ErrorId;

	tmp_ErrorEntry.ErrorText	:= ErrorPrefix;

	tmp_ErrorEntry.ErrorText	:= CONCAT(tmp_ErrorEntry.ErrorText, UDINT_TO_STRING(tmp_ErrorEntry.ErrorId));
	tmp_ErrorEntry.ErrorText	:= CONCAT(tmp_ErrorEntry.ErrorText, 'Task: ');
	tmp_ErrorEntry.ErrorText	:= CONCAT(tmp_ErrorEntry.ErrorText, MultiAxisCtrlPtr^.Input.Parameter.ThreadName);	
	tmp_ErrorEntry.ErrorText	:= CONCAT(tmp_ErrorEntry.ErrorText, FC_NcErrorMsg(tmp_ErrorEntry.ErrorId));	
	fnLogMsg(ADR(LogMsg_0),LOG_ERROR,tmp_ErrorEntry.ErrorText,0,0,0);	
	
	tmp_ErrorEntry.MotorEvents := CreateNCErrMsgDetails(tmp_ErrorEntry.ErrorId);
	
	BasicAxisCtrlPtr^.Output.Error.fbErrorHandler.ErrorPush(tmp_ErrorEntry);
END_METHOD

METHOD PRIVATE CamIn 
VAR_INPUT
END_VAR

VAR_INST
	IntErrorTrig_0 : Trigger ;
	IntErrorTrig_1 : Trigger ;
END_VAR

(*
fbMC_CamIn.MasterOffset 	:= MultiAxisCtrlPtr^.Input.Parameter.CamIn.MasterOffset;
fbMC_CamIn.SlaveOffset 		:= MultiAxisCtrlPtr^.Input.Parameter.CamIn.SlaveOffset; 
fbMC_CamIn.MasterScaling	:= MultiAxisCtrlPtr^.Input.Parameter.CamIn.MasterScaling;
fbMC_CamIn.SlaveScaling 	:= MultiAxisCtrlPtr^.Input.Parameter.CamIn.SlaveScaling;
fbMC_CamIn.StartMode 		:= MultiAxisCtrlPtr^.Input.Parameter.CamIn.StartMode;
fbMC_CamIn.CamTableID 		:= MultiAxisCtrlPtr^.Input.Parameter.CamIn.CamTableID;
fbMC_CamIn.BufferMode 		:= MultiAxisCtrlPtr^.Input.Parameter.CamIn.BufferMode;
fbMC_CamIn.Options 			:= MultiAxisCtrlPtr^.Input.Parameter.CamIn.Options; 

fbMC_CamIn.Execute := TRUE;

IF (MultiAxisCtrlPtr^.Input.Command.CamIn.DisengageSlave = TRUE) THEN
	CamIn := FALSE ;
	MultiAxisCtrlPtr^.Input.Command.CamIn.DisengageSlave := FALSE;
	MultiAxisCtrlPtr^.Output.Status.CamOut.Done := FALSE ;
	fbMC_CamIn.Execute := FALSE;
	AxisStep := MultiAxis_STATE_CAM_STOP ;
ELSE
	CamIn := TRUE ;
	AxisStep := MultiAxis_STATE_READY ;
END_IF
*)

(* check if error occured *)
IF IntErrorTrig_0.EDGEPOS(fbMC_CamIn.Error = TRUE) THEN
	// Add FB Error to ErrorHandler

	AddNCError(fbMC_CamIn.ErrorID,' NC Error fbMC_CamIn ErrorID: ');
	//Log			
	fbMC_CamIn.Execute := FALSE;
	AxisStep := MultiAxis_STATE_ERROR;
END_IF

(* check if Command Aborted occured *)
IF IntErrorTrig_1.EDGEPOS(fbMC_CamIn.CommandAborted = TRUE) THEN
	// Add PLCopen FB Error
	//Log			
	fbMC_CamIn.Execute := FALSE;
END_IF
{warning disable C0371}
//Warning: Access to VAR_IN_OUT <Var> declared in <POU> from external context <Method/Transition/Property>
fbMC_CamIn(Master := MasterRef , Slave := AxisRef);
{warning restore C0371}


MultiAxisCtrlPtr^.Output.Status.CamIn.Busy := fbMC_CamIn.Busy ;
MultiAxisCtrlPtr^.Output.Status.CamIn.CommandAborted := fbMC_CamIn.CommandAborted ;
MultiAxisCtrlPtr^.Output.Status.CamIn.InSync := fbMC_CamIn.InSync ;
MultiAxisCtrlPtr^.Output.Status.CamIn.Active := fbMC_CamIn.Active ;
END_METHOD

METHOD PRIVATE CamOut : BOOL
VAR_INPUT
END_VAR
VAR_INST
	IntErrorTrig_0 : Trigger ;
	IntErrorTrig_1 : Trigger ;
END_VAR
CamOut := FALSE ;
fbMC_CamOut.Execute := TRUE;
//fbMC_CamOut.Options := MultiAxisCtrlPtr^.Input.Parameter.CamOut.Options ;
MultiAxisCtrlPtr^.Output.Status.CamOut.Done := FALSE ;

(* check if coupling is stopped *)
IF (fbMC_CamOut.Done = TRUE) THEN
	MultiAxisCtrlPtr^.Output.Status.CamOut.Done := TRUE ;
	fbMC_CamOut.Execute := FALSE;
	CamOut := TRUE ;
	//AxisStep := MultiAxis_STATE_READY;
END_IF

(* check if error occured *)
IF IntErrorTrig_0.EDGEPOS(fbMC_CamOut.Error = TRUE) THEN
	// Add FB Error to ErrorHandler

	AddNCError(fbMC_CamOut.ErrorID,' NC Error fbMC_CamOut ErrorID: ');
	//Log
		
	fbMC_CamOut.Execute := FALSE;
	AxisStep := MultiAxis_STATE_ERROR;
END_IF
	
(* MC_CAMOUT FB Call *)
{warning disable C0371}
//Warning: Access to VAR_IN_OUT <Var> declared in <POU> from external context <Method/Transition/Property>
fbMC_CamOut(Slave := AxisRef);
{warning restore C0371}

MultiAxisCtrlPtr^.Output.Status.CamOut.Busy := fbMC_CamOut.Busy ;
END_METHOD

METHOD PRIVATE CamTableSelect : BOOL
VAR_INPUT
END_VAR
VAR_INST
	IntErrorTrig_0 : Trigger ;
	IntErrorTrig_1 : Trigger ;
END_VAR
CamTableSelect := FALSE ;
fbMC_CamTableSelect.Execute := TRUE;
//fbMC_CamTableSelect.CamTable 		:= MultiAxisCtrlPtr^.Input.Parameter.CamTableSelect.CamTable ;
fbMC_CamTableSelect.CamTableID 		:= MultiAxisCtrlPtr^.Input.Parameter.CamTableSelect.CamTableID ;
fbMC_CamTableSelect.Periodic 		:= MultiAxisCtrlPtr^.Input.Parameter.CamTableSelect.Periodic ;
fbMC_CamTableSelect.MasterAbsolute 	:= MultiAxisCtrlPtr^.Input.Parameter.CamTableSelect.MasterAbsolute ;
fbMC_CamTableSelect.SlaveAbsolute 	:= MultiAxisCtrlPtr^.Input.Parameter.CamTableSelect.SlaveAbsolute ;

MultiAxisCtrlPtr^.Output.Status.CamTableSelect.Done := FALSE ;

(* wait for CamTableSelect done *)
IF (fbMC_CamTableSelect.Done = TRUE) THEN
	CamTableSelect := TRUE ;
	MultiAxisCtrlPtr^.Output.Status.CamTableSelect.Done := TRUE ;
	fbMC_CamTableSelect.Execute := FALSE;
	//AxisStep := MultiAxis_STATE_READY;
END_IF

(* check if error occured *)
IF IntErrorTrig_0.EDGEPOS(fbMC_CamTableSelect.Error = TRUE) THEN
	// Add FB Error to ErrorHandler

	AddNCError(fbMC_CamTableSelect.ErrorID,' NC Error fbMC_CamTableSelect ErrorID: ');
	//Log
		
	fbMC_CamTableSelect.Execute := FALSE;
	AxisStep := MultiAxis_STATE_ERROR;
END_IF 

(********************** MC_CAMTABLESELECT FB Call *************************)
{warning disable C0371}
//Warning: Access to VAR_IN_OUT <Var> declared in <POU> from external context <Method/Transition/Property>
fbMC_CamTableSelect(Master := MasterRef,Slave := AxisRef,CamTable := MultiAxisCtrlPtr^.Input.Parameter.CamTableSelect.CamTable);
{warning restore C0371}

MultiAxisCtrlPtr^.Output.Status.CamTableSelect.Busy := fbMC_CamTableSelect.Busy ;
END_METHOD

METHOD PRIVATE Disable_All_FB : BOOL
VAR_INPUT
	Execute: 	BOOL;
END_VAR

VAR_INST
	DisableAllTrig: 		Trigger ;	
	DisableAllState:      USINT;   
END_VAR
IF DisableAllTrig.EDGEPOS(Execute) THEN
	DisableAllState := 1;
	Disable_All_FB := FALSE ;
END_IF

CASE DisableAllState OF
 
		
	1:
		IF fbMC_CamIn.Active THEN		
			DisableAllState := DisableAllState +1;
		ELSE	
			DisableAllState := DisableAllState +2;
		END_IF
	2:
		IF CamOut() THEN
			DisableAllState := DisableAllState +1;
		END_IF
		
	3:
		IF fbMC_GearInDyn.Active OR fbMC_GearInPos.Active OR fbMC_GearInMultiMaster.Active THEN
			DisableAllState := DisableAllState +1;
		ELSE	
			DisableAllState := DisableAllState +2;
		END_IF
	4:
		IF GearOut() THEN
			DisableAllState := DisableAllState +1;
		END_IF

	5:
		fbMC_CamOut.Execute 			:= fbMC_CamIn.Active   ;
		fbMC_CamTableSelect.Execute 	:= FALSE ;
		fbMC_CamIn.Execute 				:= FALSE ;
		
		fbMC_GearOut.Execute 			:= FALSE ;
		fbMC_GearInDyn.Enable 			:= FALSE ;				
		fbMC_GearInPos.Execute 			:= FALSE ;				
		fbMC_GearInMultiMaster.Enable	:= FALSE;
		
		{warning disable C0371}
		//Warning: Access to VAR_IN_OUT <Var> declared in <POU> from external context <Method/Transition/Property>
		fbMC_CamTableSelect(Master := MasterRef,Slave := AxisRef,CamTable := MultiAxisCtrlPtr^.Input.Parameter.CamTableSelect.CamTable);
		fbMC_CamIn(Master := MasterRef , Slave := AxisRef);
		fbMC_CamOut(Slave := AxisRef);
		fbMC_GearInDyn(Master := MasterRef , Slave := AxisRef);
		fbMC_GearInPos(Master := MasterRef , Slave := AxisRef);
		fbMC_GearOut(Slave := AxisRef);
		fbMC_GearInMultiMaster(Master1:= MasterRef, Master2:= MasterRef2, Master3:= MasterRef3, Master4:= MasterRef4, Slave:= AxisRef); 
		{warning restore C0371}
		

		
		memset(ADR(MultiAxisCtrlPtr^.Input.Command) ,0 ,SIZEOF(MultiAxisCtrlPtr^.Input.Command));
		memset(ADR(MultiAxisCtrlPtr^.Output.Status) ,0 ,SIZEOF(MultiAxisCtrlPtr^.Output.Status));
		
		Disable_All_FB := TRUE ;
	
END_CASE
END_METHOD

METHOD PRIVATE GearInDyn : BOOL
VAR_INPUT
END_VAR

VAR

END_VAR

VAR_INST
	IntErrorTrig_0 : Trigger ;
	IntErrorTrig_1 : Trigger ;
END_VAR
//GearInDyn := FALSE ;

fbMC_GearInDyn.Acceleration := MultiAxisCtrlPtr^.Input.Parameter.GearInDyn.Acceleration;
fbMC_GearInDyn.Deceleration := MultiAxisCtrlPtr^.Input.Parameter.GearInDyn.Deceleration;
fbMC_GearInDyn.GearRatio 	:= MultiAxisCtrlPtr^.Input.Parameter.GearInDyn.GearRatio;
fbMC_GearInDyn.Jerk 		:= MultiAxisCtrlPtr^.Input.Parameter.GearInDyn.Jerk;
fbMC_GearInDyn.BufferMode 	:= MultiAxisCtrlPtr^.Input.Parameter.GearInDyn.BufferMode;
fbMC_GearInDyn.Options 		:= MultiAxisCtrlPtr^.Input.Parameter.GearInDyn.Options;

IF MultiAxisCtrlPtr^.Input.Command.GearInDyn.DisengageSlave THEN
	MultiAxisCtrlPtr^.Input.Command.GearInDyn.StartSlave := FALSE ;
	fbMC_GearInDyn.Enable := FALSE ;
	GearInDyn := FALSE ;
ELSE
	fbMC_GearInDyn.Enable := TRUE ;	
END_IF

(* check if error occured *)
IF IntErrorTrig_0.EDGEPOS(fbMC_GearInDyn.Error = TRUE) THEN
	// Add FB Error to ErrorHandler
	
	AddNCError(fbMC_GearInDyn.ErrorID,' NC Error fbMC_GearInDyn ErrorID: ');
	
	//Log			
	fbMC_GearInDyn.Enable 	:= FALSE;
	GearInDyn := FALSE ;
	AxisStep 				:= MultiAxis_STATE_ERROR;
END_IF

(* check if Command Aborted occured *)
IF IntErrorTrig_1.EDGEPOS(fbMC_GearInDyn.CommandAborted = TRUE) THEN
	// Add PLCopen FB Error
	//Log	
	fbMC_GearInDyn.Enable 	:= FALSE;
	GearInDyn := FALSE ;
	AxisStep 				:= MultiAxis_STATE_READY;
END_IF
{warning disable C0371}
//Warning: Access to VAR_IN_OUT <Var> declared in <POU> from external context <Method/Transition/Property>
fbMC_GearInDyn(Master := MasterRef , Slave := AxisRef ) ;
{warning restore C0371}


MultiAxisCtrlPtr^.Output.Status.GearInDyn.Active 			:= fbMC_GearInDyn.Active;
MultiAxisCtrlPtr^.Output.Status.GearInDyn.Busy 				:= fbMC_GearInDyn.Busy;
MultiAxisCtrlPtr^.Output.Status.GearInDyn.CommandAborted 	:= fbMC_GearInDyn.CommandAborted;
MultiAxisCtrlPtr^.Output.Status.GearInDyn.InGear 			:= fbMC_GearInDyn.InGear;

IF tempTrig.EDGEPOS(fbMC_GearInDyn.InGear) THEN
	GearInDyn := TRUE ;	
END_IF
END_METHOD

METHOD PRIVATE GearInMultiMaster : BOOL
VAR_INPUT
END_VAR

VAR

END_VAR

VAR_INST
	IntErrorTrig_0 : Trigger ;
	IntErrorTrig_1 : Trigger ;
END_VAR
//GearInMultiMaster := FALSE ;
GearInMultiMaster:= fbMC_GearInMultiMaster.InGear ;
fbMC_GearInMultiMaster.Acceleration := MultiAxisCtrlPtr^.Input.Parameter.GearInMultiMaster.Acceleration;
fbMC_GearInMultiMaster.Deceleration := MultiAxisCtrlPtr^.Input.Parameter.GearInMultiMaster.Deceleration;
fbMC_GearInMultiMaster.GearRatio1 	:= MultiAxisCtrlPtr^.Input.Parameter.GearInMultiMaster.GearRatio1;
fbMC_GearInMultiMaster.GearRatio2 	:= MultiAxisCtrlPtr^.Input.Parameter.GearInMultiMaster.GearRatio2;
fbMC_GearInMultiMaster.GearRatio3 	:= MultiAxisCtrlPtr^.Input.Parameter.GearInMultiMaster.GearRatio3;
fbMC_GearInMultiMaster.GearRatio4 	:= MultiAxisCtrlPtr^.Input.Parameter.GearInMultiMaster.GearRatio4;
fbMC_GearInMultiMaster.Jerk 		:= MultiAxisCtrlPtr^.Input.Parameter.GearInMultiMaster.Jerk;
fbMC_GearInMultiMaster.BufferMode 	:= MultiAxisCtrlPtr^.Input.Parameter.GearInMultiMaster.BufferMode;
fbMC_GearInMultiMaster.Options 		:= MultiAxisCtrlPtr^.Input.Parameter.GearInMultiMaster.Options;

IF (MultiAxisCtrlPtr^.Input.Command.GearInMultiMaster.DisengageSlave) 
	OR BasicAxisCtrlPtr^.Input.Command.Power = FALSE THEN
	MultiAxisCtrlPtr^.Input.Command.GearInMultiMaster.StartSlave := FALSE;
	fbMC_GearInMultiMaster.Enable := FALSE ;
	//GearInMultiMaster := FALSE ;
ELSE
	fbMC_GearInMultiMaster.Enable := TRUE ;	
	GearInMultiMaster := TRUE;
END_IF

(* check if error occured *)
IF IntErrorTrig_0.EDGEPOS(fbMC_GearInMultiMaster.Error = TRUE) THEN
	// Add FB Error to ErrorHandler
	
	AddNCError(fbMC_GearInMultiMaster.ErrorID,' NC Error fbMC_GearInMultiMaster ErrorID: ');
	//Log			
	fbMC_GearInMultiMaster.Enable 	:= FALSE;
	GearInMultiMaster := FALSE ;
	AxisStep 				:= MultiAxis_STATE_ERROR;
END_IF

(* check if Command Aborted occured *)
IF IntErrorTrig_1.EDGEPOS(fbMC_GearInMultiMaster.CommandAborted = TRUE) THEN
	// Add PLCopen FB Error
	//Log	
	fbMC_GearInMultiMaster.Enable 	:= FALSE;
	GearInMultiMaster := FALSE ;
	AxisStep 				:= MultiAxis_STATE_READY;
END_IF

{warning disable C0371}
//Warning: Access to VAR_IN_OUT <Var> declared in <POU> from external context <Method/Transition/Property>
fbMC_GearInMultiMaster(Master1:= MasterRef, Master2:= MasterRef2, Master3:= MasterRef3, Master4:= MasterRef4, Slave:= AxisRef); 
{warning restore C0371}


MultiAxisCtrlPtr^.Output.Status.GearInMultiMaster.Active 			:= fbMC_GearInMultiMaster.Active;
MultiAxisCtrlPtr^.Output.Status.GearInMultiMaster.Busy 				:= fbMC_GearInMultiMaster.Busy;
MultiAxisCtrlPtr^.Output.Status.GearInMultiMaster.CommandAborted 	:= fbMC_GearInMultiMaster.CommandAborted;
MultiAxisCtrlPtr^.Output.Status.GearInMultiMaster.InGear 			:= fbMC_GearInMultiMaster.InGear;

//IF tempTrig.EDGEPOS(fbMC_GearInMultiMaster.InGear) THEN
//	GearInMultiMaster := TRUE ;	
//END_IF
END_METHOD

METHOD PRIVATE GearInPos : BOOL
VAR_INPUT
END_VAR
VAR_INST
	IntErrorTrig_0 : Trigger ;
	IntErrorTrig_1 : Trigger ;
END_VAR

fbMC_GearInPos.Acceleration 			:= MultiAxisCtrlPtr^.Input.Parameter.GearInPos.Acceleration;
fbMC_GearInPos.Deceleration 			:= MultiAxisCtrlPtr^.Input.Parameter.GearInPos.Deceleration;
fbMC_GearInPos.MasterStartDistance 		:= MultiAxisCtrlPtr^.Input.Parameter.GearInPos.MasterStartDistance;
fbMC_GearInPos.MasterSyncPosition 		:= MultiAxisCtrlPtr^.Input.Parameter.GearInPos.MasterSyncPosition;
fbMC_GearInPos.SlaveSyncPosition 		:= MultiAxisCtrlPtr^.Input.Parameter.GearInPos.SlaveSyncPosition;
fbMC_GearInPos.RatioDenominator 		:= MultiAxisCtrlPtr^.Input.Parameter.GearInPos.RatioDenominator;
fbMC_GearInPos.RatioNumerator 			:= MultiAxisCtrlPtr^.Input.Parameter.GearInPos.RatioNumerator;
fbMC_GearInPos.SyncMode					:= MultiAxisCtrlPtr^.Input.Parameter.GearInPos.SyncMode;
fbMC_GearInPos.Velocity					:= MultiAxisCtrlPtr^.Input.Parameter.GearInPos.Velocity;
fbMC_GearInPos.Jerk 					:= MultiAxisCtrlPtr^.Input.Parameter.GearInPos.Jerk;
fbMC_GearInPos.BufferMode 				:= MultiAxisCtrlPtr^.Input.Parameter.GearInPos.BufferMode;
//fbMC_GearInPos.Options 					:= MultiAxisCtrlPtr^.Input.Parameter.GearInPos.Options;

IF MultiAxisCtrlPtr^.Input.Command.GearInPos.DisengageSlave THEN
	GearInPos := FALSE ;
	fbMC_GearInPos.Execute := FALSE ;
ELSIF NOT MultiAxisCtrlPtr^.Output.Status.GearInPos.InSync THEN
	fbMC_GearInPos.Execute := TRUE ;	
END_IF

(* check if error occured *)
IF IntErrorTrig_0.EDGEPOS(fbMC_GearInPos.Error = TRUE) THEN
	// Add FB Error to ErrorHandler
	AddNCError(fbMC_GearInPos.ErrorID,' NC Error fbMC_GearInPos ErrorID: ');

	//Log	
	fbMC_GearInPos.Execute 	:= FALSE;
	GearInPos := FALSE ;
	AxisStep 				:= MultiAxis_STATE_ERROR;
END_IF

(* check if Command Aborted occured *)
IF IntErrorTrig_1.EDGEPOS(fbMC_GearInPos.CommandAborted = TRUE) THEN
	// Add PLCopen FB Error
	//Log		
	fbMC_GearInPos.Execute 	:= FALSE;
	GearInPos := FALSE ;
	AxisStep 				:= MultiAxis_STATE_READY;
END_IF
{warning disable C0371}
//Warning: Access to VAR_IN_OUT <Var> declared in <POU> from external context <Method/Transition/Property>
fbMC_GearInPos(Slave:= AxisRef , Master := MasterRef ) ;
{warning restore C0371}


MultiAxisCtrlPtr^.Output.Status.GearInPos.Active 			:= fbMC_GearInPos.Active;
MultiAxisCtrlPtr^.Output.Status.GearInPos.Busy 				:= fbMC_GearInPos.Busy;
MultiAxisCtrlPtr^.Output.Status.GearInPos.CommandAborted 	:= fbMC_GearInPos.CommandAborted;
MultiAxisCtrlPtr^.Output.Status.GearInPos.InSync 			:= fbMC_GearInPos.InSync;
MultiAxisCtrlPtr^.Output.Status.GearInPos.StartSync 		:= fbMC_GearInPos.StartSync;

IF tempTrig.EDGEPOS(MultiAxisCtrlPtr^.Output.Status.GearInPos.InSync) THEN
	GearInPos := TRUE ;
END_IF
END_METHOD

METHOD PRIVATE GearOut : BOOL
VAR_INPUT
END_VAR
VAR_INST
	IntErrorTrig_0 : Trigger ;
	IntErrorTrig_1 : Trigger ;
END_VAR
//fbMC_GearOut.Options 			:= MultiAxisCtrlPtr^.Input.Parameter.GearOut.Options;
GearOut := FALSE ;
fbMC_GearOut.Execute := TRUE ;	
MultiAxisCtrlPtr^.Input.Command.GearInDyn.DisengageSlave := FALSE ;
MultiAxisCtrlPtr^.Input.Command.GearInPos.DisengageSlave := FALSE ;
MultiAxisCtrlPtr^.Input.Command.GearInMultiMaster.DisengageSlave := FALSE ;

(* check if error occured *)
IF IntErrorTrig_0.EDGEPOS(fbMC_GearOut.Error = TRUE) THEN
	// Add FB Error to ErrorHandler
	AddNCError(fbMC_GearOut.ErrorID,' NC Error fbMC_GearOut ErrorID: ');
	
	//Log	
	fbMC_GearOut.Execute 	:= FALSE;
	GearOut := FALSE ;
	AxisStep 				:= MultiAxis_STATE_ERROR;
END_IF

IF (fbMC_GearOut.Done) THEN
	MultiAxisCtrlPtr^.Output.Status.GearOut.Done 	:= TRUE ;
	fbMC_GearOut.Execute 	:= FALSE;
	GearOut := TRUE ;
END_IF

{warning disable C0371}
//Warning: Access to VAR_IN_OUT <Var> declared in <POU> from external context <Method/Transition/Property>
fbMC_GearOut(Slave := AxisRef) ;
{warning restore C0371}



MultiAxisCtrlPtr^.Output.Status.GearOut.Busy 	:= fbMC_GearOut.Busy;
//MultiAxisCtrlPtr^.Output.Status.GearOut.Done 	:= fbMC_GearOut.Done;
END_METHOD

METHOD PRIVATE ResetAll_MC_FB : BOOL

		fbMC_CamOut.Execute 			:= fbMC_CamIn.Active   ;
		fbMC_CamTableSelect.Execute 	:= FALSE ;
		fbMC_CamIn.Execute 				:= FALSE ;
		
		fbMC_GearOut.Execute 			:= FALSE ;
		fbMC_GearInDyn.Enable 			:= FALSE ;				
		fbMC_GearInPos.Execute 			:= FALSE ;				
		fbMC_GearInMultiMaster.Enable	:= FALSE;
		
		{warning disable C0371}
		//Warning: Access to VAR_IN_OUT <Var> declared in <POU> from external context <Method/Transition/Property>
		fbMC_CamTableSelect(Master := MasterRef,Slave := AxisRef,CamTable := MultiAxisCtrlPtr^.Input.Parameter.CamTableSelect.CamTable);
		fbMC_CamIn(Master := MasterRef , Slave := AxisRef);
		fbMC_CamOut(Slave := AxisRef);
		fbMC_GearInDyn(Master := MasterRef , Slave := AxisRef);
		fbMC_GearInPos(Master := MasterRef , Slave := AxisRef);
		fbMC_GearOut(Slave := AxisRef);
		fbMC_GearInMultiMaster(Master1:= MasterRef, Master2:= MasterRef2, Master3:= MasterRef3, Master4:= MasterRef4, Slave:= AxisRef); 
		{warning restore C0371}
		

		
		memset(ADR(MultiAxisCtrlPtr^.Input.Command) ,0 ,SIZEOF(MultiAxisCtrlPtr^.Input.Command));
		memset(ADR(MultiAxisCtrlPtr^.Output.Status) ,0 ,SIZEOF(MultiAxisCtrlPtr^.Output.Status));
		
		ResetAll_MC_FB := TRUE ;
END_METHOD

END_FUNCTION_BLOCK

// ---- POUs/Lib/Motion/CyclicAxis_FB.TcPOU
FUNCTION_BLOCK PUBLIC CyclicAxis_FB
VAR_INPUT
	
	BasicAxisCtrlPtr 	: POINTER TO Basic_axis_typ ;
	CyclicAxisCtrlPtr 	: POINTER TO CyclicAxis_typ ;
	
END_VAR
VAR_IN_OUT
	
	AxisRef		: 	AXIS_REF;
END_VAR
VAR_OUTPUT
END_VAR
	
VAR
	LogMsgInit		: BOOL;
	LogMsg_0 		: LogMsg ;
	
//	GetCycleTime:	FB_CTRL_GET_TASK_CYCLETIME;
//	CycleTime:		TIME;
//	CycleTimeInit:	BOOL;
	
	
	fbGetCurTaskIdx: 		GETCURTASKINDEX;
    TaskCycleTimeUDINT: 	UDINT;
    TaskCycleTime: 			TIME;

	
	
	DisableTriger	: Trigger ;
	Disable			: BOOL ;
	
	fbMC_PositionCorrectionLimiter:	MC_PositionCorrectionLimiter;
		
	fbMC_ExtSetPointGenEnable:		MC_ExtSetPointGenEnable;	
	fbMC_ExtSetPointGenDisable:		MC_ExtSetPointGenDisable;
	
	
	ErrorTrig : Trigger ;
	AxisStep : eCyclicAxisState ;
	
	tmp_ErrorEntry			: Eh_ErrorEntry_typ;
END_VAR

IF NOT LogMsgInit THEN
	LogMsgInit	:= TRUE;
	LogMsg_0.logData.category	:= BasicAxisCtrlPtr^.Input.Parameter.ThreadName;
	LogMsg_0.ptrGlobalArray		:= ADR(LogGlobalArray);
	LogMsg_0.ptrEncoderAngle	:= ADR(BasicAxisCtrlPtr^.Input.Parameter.PosForLog);
	LogMsg_0.Enable				:= TRUE;
END_IF

IF (TaskCycleTimeUDINT = 0) THEN
	fbGetCurTaskIdx();
	TaskCycleTimeUDINT	:= _TaskInfo[fbGetCurTaskIdx.index].CycleTime;
	TaskCycleTime		:= UDINT_TO_TIME(TaskCycleTimeUDINT/10000);
END_IF

IF BasicAxisCtrlPtr^.Output.Status.FAULT THEN
	THIS^.ResetAll_MC_FB();
	AxisStep	:= CyclicAxis_STATE_ERROR;
END_IF

//In case of Stop go to STATE_DISABLE
IF (AxisStep = CyclicAxis_STATE_POS_ACTIVE OR AxisStep = CyclicAxis_STATE_VEL_ACTIVE)
	AND (BasicAxisCtrlPtr^.Input.Command.Stop = TRUE) OR (BasicAxisCtrlPtr^.Input.Command.Halt = TRUE) THEN
	AxisStep := CyclicAxis_STATE_DISABLE;
END_IF

CASE AxisStep OF
	(******************** WAIT *************************)
	CyclicAxis_STATE_WAIT: (* STATE: Wait *)
		IF BasicAxisCtrlPtr^.Output.Status.ReadyForCmd THEN
			AxisStep	:= CyclicAxis_STATE_READY;
		END_IF
		
		THIS^.ResetAll_MC_FB();
		
	(******************** READY *************************)
	CyclicAxis_STATE_READY:
		IF CyclicAxisCtrlPtr^.Input.Command.CyclicPos.Start THEN
			CyclicAxisCtrlPtr^.Input.Command.CyclicPos.Start	:= FALSE ;
			AxisStep	:= CyclicAxis_STATE_POS_ACTIVE;
		ELSIF CyclicAxisCtrlPtr^.Input.Command.CyclicVel.Start THEN
			CyclicAxisCtrlPtr^.Input.Command.CyclicVel.Start	:= FALSE;
			AxisStep	:= CyclicAxis_STATE_VEL_ACTIVE;
		END_IF
		
	(******************** Cyclic Pos Active **********************)
	CyclicAxis_STATE_POS_ACTIVE:
		IF CyclicAxisCtrlPtr^.Input.Command.CyclicPos.Disable  THEN
			CyclicAxisCtrlPtr^.Input.Command.CyclicPos.Disable	:= FALSE;
			AxisStep	:= CyclicAxis_STATE_DISABLE;
		ELSE
			CyclicPos();
			//CyclicPosTest();
		END_IF
		
	(******************** Cyclic Vel Active **********************)
	CyclicAxis_STATE_VEL_ACTIVE:
		IF CyclicAxisCtrlPtr^.Input.Command.CyclicVel.Disable  THEN
			CyclicAxisCtrlPtr^.Input.Command.CyclicVel.Disable	:= FALSE;
			AxisStep	:= CyclicAxis_STATE_DISABLE;
		ELSE
			CyclicVel();
		END_IF
		
	(******************** Cyclic Pos Disable  **********************)
	CyclicAxis_STATE_DISABLE:
		
		IF THIS^.CyclicDisable() THEN
			AxisStep	:= CyclicAxis_STATE_READY;
		END_IF
		
	(******************** Error **********************)
	CyclicAxis_STATE_ERROR:
		THIS^.ResetAll_MC_FB();
		IF BasicAxisCtrlPtr^.Output.Status.FAULT THEN
			AxisStep	:= CyclicAxis_STATE_ERROR;
		ELSE
			CyclicAxisCtrlPtr^.Output.Error.ErrorID	:= 0;
			AxisStep	:= CyclicAxis_STATE_WAIT;
		END_IF
		
END_CASE

CyclicAxisCtrlPtr^.Output.Status.CyclicPos.Busy	:= fbMC_ExtSetPointGenEnable.Busy OR fbMC_ExtSetPointGenDisable.Busy;

IF DisableTriger.EDGEPOS(BasicAxisCtrlPtr^.Output.Status.AxisStatus.Error)THEN
	Disable	:= TRUE ;
END_IF
IF Disable THEN
	IF THIS^.CyclicDisable() THEN
		Disable	:= FALSE ;
	END_IF
END_IF

//=====================================================================================================================\\

//fnLogTransfer FUNCTION call
fnLogTransfer(ADR(LogMsg_0));

METHOD AddNCError : BOOL
VAR_INPUT
	ErrorId			: UDINT;
	ErrorPrefix     : STRING[100];
END_VAR

	tmp_ErrorEntry.ErrorId		:= ErrorId;

	tmp_ErrorEntry.ErrorText	:= ErrorPrefix;

	tmp_ErrorEntry.ErrorText	:= CONCAT(tmp_ErrorEntry.ErrorText, UDINT_TO_STRING(tmp_ErrorEntry.ErrorId));
	tmp_ErrorEntry.ErrorText	:= CONCAT(tmp_ErrorEntry.ErrorText, 'Task: ');
	tmp_ErrorEntry.ErrorText	:= CONCAT(tmp_ErrorEntry.ErrorText, CyclicAxisCtrlPtr^.Input.Parameter.ThreadName);	
	tmp_ErrorEntry.ErrorText	:= CONCAT(tmp_ErrorEntry.ErrorText, FC_NcErrorMsg(tmp_ErrorEntry.ErrorId));	
	fnLogMsg(ADR(LogMsg_0),LOG_ERROR,tmp_ErrorEntry.ErrorText,0,0,0);	
	
	tmp_ErrorEntry.MotorEvents := CreateNCErrMsgDetails(tmp_ErrorEntry.ErrorId);
	
	BasicAxisCtrlPtr^.Output.Error.fbErrorHandler.ErrorPush(tmp_ErrorEntry);
END_METHOD

METHOD PRIVATE CyclicDisable : BOOL
VAR_INPUT
END_VAR
VAR_INST
	IntErrorTrig_0:	Trigger;
END_VAR

CyclicDisable	:= FALSE ;
fbMC_ExtSetPointGenDisable.Execute	:= TRUE;
fbMC_ExtSetPointGenEnable.Execute	:= FALSE;
CyclicAxisCtrlPtr^.Input.Command.CyclicPos.Disable	:= FALSE;
CyclicAxisCtrlPtr^.Input.Command.CyclicVel.Disable	:= FALSE;

(* check if error occured *)
IF IntErrorTrig_0.EDGEPOS(fbMC_ExtSetPointGenDisable.Error = TRUE) THEN
	// Add FB Error to ErrorHandler
	AddNCError(fbMC_ExtSetPointGenDisable.ErrorID,'NC Error fbMC_ExtSetPointGenDisable ErrorID:');
	//Log
	fbMC_ExtSetPointGenDisable.Execute 	:= FALSE;
	CyclicDisable	:= FALSE ;
	AxisStep		:= CyclicAxis_STATE_ERROR;
END_IF
IF (CyclicAxisCtrlPtr^.Output.Status.CyclicPos.Active = TRUE) THEN
	CyclicAxisCtrlPtr^.Output.Status.CyclicPos.Busy	:= fbMC_ExtSetPointGenDisable.Busy;
ELSIF(CyclicAxisCtrlPtr^.Output.Status.CyclicPos.Active = TRUE) THEN
	CyclicAxisCtrlPtr^.Output.Status.CyclicVel.Busy	:= fbMC_ExtSetPointGenDisable.Busy;
END_IF

IF (fbMC_ExtSetPointGenDisable.Done
	AND fbMC_ExtSetPointGenDisable.Enabled = FALSE) THEN
	CyclicAxisCtrlPtr^.Output.Status.CyclicPos.Active	:= FALSE;
	CyclicAxisCtrlPtr^.Output.Status.CyclicVel.Active	:= FALSE;
	CyclicAxisCtrlPtr^.Output.Status.CyclicPos.Busy	:= FALSE;
	CyclicAxisCtrlPtr^.Output.Status.CyclicVel.Busy	:= FALSE;
	fbMC_ExtSetPointGenDisable.Execute 	:= FALSE;
	CyclicDisable	:= TRUE;
END_IF
{warning disable C0371}
//Warning: Access to VAR_IN_OUT <Var> declared in <POU> from external context <Method/Transition/Property>
fbMC_ExtSetPointGenDisable(Axis:= AxisRef);
fbMC_ExtSetPointGenEnable(Axis:= AxisRef);
{warning restore C0371}
END_METHOD

METHOD PRIVATE CyclicPos : BOOL
VAR_INPUT
END_VAR

VAR

END_VAR

VAR_INST
	IntErrorTrig_0 : Trigger ;
	
	fbReadParam_SWLimitPos:	MC_ReadParameter;
	fbReadParam_SWLimitNeg:	MC_ReadParameter;
	
	fbSramp_PosGen:		SrampHp;
	State:			INT;
	InitCompleted:	BOOL;
END_VAR
	
	IF fbMC_ExtSetPointGenEnable.Enabled = FALSE
		AND InitCompleted THEN
		InitCompleted	:= FALSE;
		State			:= 0;
	END_IF
	
	CASE State OF
		0: // Init
			// Initialize Velocity Generator, fbSramp
			fbSramp_PosGen.VD_MAX	:= CyclicAxisCtrlPtr^.Input.Parameter.CyclicPos.Velocity * (-1);
			fbSramp_PosGen.VU_MAX	:= CyclicAxisCtrlPtr^.Input.Parameter.CyclicPos.Velocity;
			fbSramp_PosGen.A_DN		:= CyclicAxisCtrlPtr^.Input.Parameter.CyclicPos.MaxDcc * (-1);
			fbSramp_PosGen.A_UP		:= CyclicAxisCtrlPtr^.Input.Parameter.CyclicPos.MaxAcc;
			
			//************************************************
			// Read Axis Positive SW Limit Parameter
			fbReadParam_SWLimitPos.ReadMode	:= READMODE_ONCE;
			IF NOT fbReadParam_SWLimitPos.Valid THEN
				fbReadParam_SWLimitPos.Enable	:= TRUE;
			END_IF
			fbReadParam_SWLimitPos.ParameterNumber	:= SWLimitPos;
			{warning disable C0371}
			//Warning: Access to VAR_IN_OUT <Var> declared in <POU> from external context <Method/Transition/Property>
			fbReadParam_SWLimitPos(Axis:=AxisRef);
			{warning restore C0371}
			IF fbReadParam_SWLimitPos.Valid THEN
				fbSramp_PosGen.LIMIT_HIGH	:= fbReadParam_SWLimitPos.Value;
			END_IF
			//**************************************************
			// Read Axis Negative SW Limit Parameter
			fbReadParam_SWLimitNeg.ReadMode		:= READMODE_ONCE;
			IF NOT fbReadParam_SWLimitNeg.Valid THEN
				fbReadParam_SWLimitNeg.Enable	:= TRUE;
			END_IF
			fbReadParam_SWLimitNeg.ParameterNumber	:= SWLimitNeg;
			{warning disable C0371}
			//Warning: Access to VAR_IN_OUT <Var> declared in <POU> from external context <Method/Transition/Property>
			fbReadParam_SWLimitNeg(Axis	:= AxisRef);
			{warning restore C0371}
			IF fbReadParam_SWLimitNeg.Valid THEN
				fbSramp_PosGen.LIMIT_LOW	:= fbReadParam_SWLimitNeg.Value;
			END_IF
			
			// Initialize Position to Actual Position
			fbSramp_PosGen.X	:= BasicAxisCtrlPtr^.Output.monitor.ActPosition;
			fbSramp_PosGen.SET	:= TRUE;
			fbSramp_PosGen();
			
			IF fbReadParam_SWLimitNeg.Valid
				AND fbReadParam_SWLimitPos.Valid THEN
				fbSramp_PosGen.SET	:= FALSE;
				
				{warning disable C0371}
				//Warning: Access to VAR_IN_OUT <Var> declared in <POU> from external context <Method/Transition/Property>
				AxisRef.PlcToNc.ExtSetDirection	:= 1;
				AxisRef.PlcToNc.ExtSetPos		:= fbSramp_PosGen.Y;
				{warning restore C0371}
	
				// Enable External Set Position
				fbMC_ExtSetPointGenEnable.Execute	:= TRUE;
				
				State	:= 10;
			END_IF
			
			
		10: // Wait External Set Position Enabled
			fbSramp_PosGen();
		 	IF fbMC_ExtSetPointGenEnable.Enabled THEN
				InitCompleted	:= TRUE;
				CyclicPos		:= TRUE;
				State	:= 20;
			ELSIF fbMC_ExtSetPointGenEnable.Execute = FALSE THEN
				InitCompleted	:= FALSE;
				CyclicPos		:= FALSE;
				State	:= 0; // Init	
			END_IF
			
		20: // Cyclic Position Active
			
			// Copy Velocity Generator parameters, fbSramp
			fbSramp_PosGen.VD_MAX	:= CyclicAxisCtrlPtr^.Input.Parameter.CyclicPos.Velocity * (-1);
			fbSramp_PosGen.VU_MAX	:= CyclicAxisCtrlPtr^.Input.Parameter.CyclicPos.Velocity;
			fbSramp_PosGen.A_DN		:= CyclicAxisCtrlPtr^.Input.Parameter.CyclicPos.MaxDcc * (-1);
			fbSramp_PosGen.A_UP		:= CyclicAxisCtrlPtr^.Input.Parameter.CyclicPos.MaxAcc;
			
			// Call Position Generator with new set point, SRAMP
			fbSramp_PosGen.X	:= LREAL_TO_REAL(CyclicAxisCtrlPtr^.Input.Parameter.CyclicPos.SetPos);
			fbSramp_PosGen();
			
			// Copy Integrator Output to ExtSetPos
			{warning disable C0371}
			//Warning: Access to VAR_IN_OUT <Var> declared in <POU> from external context <Method/Transition/Property>
			AxisRef.PlcToNc.ExtSetDirection	:= 1;
			AxisRef.PlcToNc.ExtSetPos		:= fbSramp_PosGen.Y;
			{warning restore C0371}
			
	END_CASE
	
	// Call External Set Position function block
	{warning disable C0371}
	//Warning: Access to VAR_IN_OUT <Var> declared in <POU> from external context <Method/Transition/Property>
	fbMC_ExtSetPointGenEnable(Axis:= AxisRef); 
	{warning restore C0371}
	
	(* check if error occured *)
	IF IntErrorTrig_0.EDGEPOS(fbMC_ExtSetPointGenEnable.Error = TRUE) THEN
		// Add FB Error to ErrorHandler
		AddNCError(fbMC_ExtSetPointGenEnable.ErrorID, 'NC Error fbMC_ExtSetPointGenEnable ErrorID:');
		
		fbMC_ExtSetPointGenEnable.Execute	:= FALSE;
		CyclicPos	:= FALSE;
		AxisStep	:= CyclicAxis_STATE_ERROR;
	END_IF


	CyclicAxisCtrlPtr^.Output.Status.CyclicPos.Active	:= fbMC_ExtSetPointGenEnable.Enabled;
	CyclicAxisCtrlPtr^.Output.Status.CyclicPos.Busy		:= fbMC_ExtSetPointGenEnable.Busy;
END_METHOD

METHOD CyclicPosTest : BOOL
VAR_INPUT
END_VAR
CyclicPosTest := FALSE ;


fbMC_PositionCorrectionLimiter.PositionCorrectionValue:= 	CyclicAxisCtrlPtr^.Input.Parameter.CyclicPos.SetPos; 
fbMC_PositionCorrectionLimiter.Acceleration:= 				CyclicAxisCtrlPtr^.Input.Parameter.CyclicPos.MaxAcc;
fbMC_PositionCorrectionLimiter.CorrectionMode:= 			POSITIONCORRECTION_MODE_FAST;
fbMC_PositionCorrectionLimiter.CorrectionLength:=			360000;
{warning disable C0371}
//Warning: Access to VAR_IN_OUT <Var> declared in <POU> from external context <Method/Transition/Property>
fbMC_PositionCorrectionLimiter(Axis := AxisRef);
{warning restore C0371}




(* check if error occured *)
IF errorTrig.EDGEPOS(fbMC_PositionCorrectionLimiter.Error) THEN
	
	// Add FB Error to ErrorHandler
	AddNCError(fbMC_PositionCorrectionLimiter.ErrorID,'NC Error fbMC_PositionCorrectionLimiter ErrorID:');	
	CyclicPosTest :=  FALSE ;
	fbMC_PositionCorrectionLimiter.Enable:= FALSE;
END_IF


CyclicAxisCtrlPtr^.Output.Status.CyclicPos.Busy:= 	fbMC_PositionCorrectionLimiter.Busy ;
CyclicAxisCtrlPtr^.Output.Status.CyclicPos.Active:= fbMC_PositionCorrectionLimiter.Limiting;
END_METHOD

METHOD PRIVATE CyclicVel : BOOL
VAR_INPUT
END_VAR

VAR

END_VAR

VAR_INST
	IntErrorTrig_0:				Trigger;
	
	fbVelocityIntegrator:		FB_CTRL_I;
	VelocityIntegratorParams:	ST_CTRL_I_PARAMS;
	
	fbReadParam_SWLimitPos:		MC_ReadParameter;
	fbReadParam_SWLimitNeg:		MC_ReadParameter;
	
	fbSrampVelocityProfile:		SrampHp;
	State:			INT;
	InitCompleted:	BOOL;
	
	
END_VAR
	
	IF fbMC_ExtSetPointGenEnable.Enabled = FALSE
		AND InitCompleted THEN
		InitCompleted	:= FALSE;
		State			:= 0;
		
	END_IF
	
	CASE State OF
		0: // Init
			fbVelocityIntegrator.bSync		:= FALSE;
			fbVelocityIntegrator(stParams	:= VelocityIntegratorParams);
			State			:= 1;
		1: 
			// Initialize Velocity Generator, fbSramp
			fbSrampVelocityProfile.VU_MAX	:= LREAL_TO_REAL(CyclicAxisCtrlPtr^.Input.Parameter.CyclicVel.MaxAcc);
			fbSrampVelocityProfile.VD_MAX	:= LREAL_TO_REAL(CyclicAxisCtrlPtr^.Input.Parameter.CyclicVel.MaxDcc * (-1));
			fbSrampVelocityProfile.A_UP		:= LREAL_TO_REAL(CyclicAxisCtrlPtr^.Input.Parameter.CyclicVel.Jerk);
			fbSrampVelocityProfile.A_DN		:= LREAL_TO_REAL(CyclicAxisCtrlPtr^.Input.Parameter.CyclicVel.Jerk * (-1));
	
			fbSrampVelocityProfile.LIMIT_HIGH	:= 1E38; 
			fbSrampVelocityProfile.LIMIT_LOW	:= -1E38;	
			
			// Initialize Velocity to Actual Velocity
			fbSrampVelocityProfile.X	:= BasicAxisCtrlPtr^.Output.monitor.ActVelocity;
			fbSrampVelocityProfile.SET	:= TRUE;
			fbSrampVelocityProfile();
			
			// Initialize Integrator for Position Generation
			VelocityIntegratorParams.fOutMaxLimit		:= 1E38;
			VelocityIntegratorParams.fOutMinLimit		:= -1E38;
			VelocityIntegratorParams.tCtrlCycleTime		:= TaskCycleTime;  
			VelocityIntegratorParams.tTaskCycleTime		:= TaskCycleTime;  
			VelocityIntegratorParams.tTi				:= T#1S;
			
			// Initialize Integrator with Actual Position
			fbVelocityIntegrator.fIn			:= fbSrampVelocityProfile.Y;
			fbVelocityIntegrator.fManSyncValue	:= BasicAxisCtrlPtr^.Output.monitor.ActPosition;
			fbVelocityIntegrator.eMode			:= eCTRL_MODE_ACTIVE;
			fbVelocityIntegrator.bSync			:= TRUE;
			fbVelocityIntegrator(stParams	:= VelocityIntegratorParams);
			
			IF fbVelocityIntegrator.fOut = fbVelocityIntegrator.fManSyncValue THEN
				fbSrampVelocityProfile.SET	:= FALSE;
				fbVelocityIntegrator.bSync	:= FALSE;
				
				
				{warning disable C0371}
				//Warning: Access to VAR_IN_OUT <Var> declared in <POU> from external context <Method/Transition/Property>
				AxisRef.PlcToNc.ExtSetDirection	:= 1;
				AxisRef.PlcToNc.ExtSetPos		:= fbVelocityIntegrator.fOut;
				{warning restore C0371}
	
				// Enable External Set Position
				fbMC_ExtSetPointGenEnable.Execute	:= TRUE;
				
				State	:= 10;
			END_IF
			
			
		10: // Wait External Set Position Enabled
		 	IF fbMC_ExtSetPointGenEnable.Enabled THEN
				InitCompleted	:= TRUE;
				CyclicVel		:= TRUE ;
				State	:= 20;
				
			ELSIF fbMC_ExtSetPointGenEnable.Execute = FALSE THEN
				InitCompleted	:= FALSE;
				CyclicVel		:= FALSE;
				fbVelocityIntegrator.bSync		:= FALSE;
				fbVelocityIntegrator(stParams	:= VelocityIntegratorParams);
				State	:= 0; // Init
			END_IF
			
		20: // Cyclic Velocity Active
			// Limit Velocity
			IF ABS(CyclicAxisCtrlPtr^.Input.Parameter.CyclicVel.SetVel) > CyclicAxisCtrlPtr^.Input.Parameter.CyclicVel.MaxVelocity THEN
				IF CyclicAxisCtrlPtr^.Input.Parameter.CyclicVel.SetVel >= 0 THEN
					fbSrampVelocityProfile.X	:= LREAL_TO_REAL(CyclicAxisCtrlPtr^.Input.Parameter.CyclicVel.MaxVelocity);
				ELSE
					fbSrampVelocityProfile.X	:= LREAL_TO_REAL( -CyclicAxisCtrlPtr^.Input.Parameter.CyclicVel.MaxVelocity);
				END_IF
			ELSE
				fbSrampVelocityProfile.X	:= LREAL_TO_REAL(CyclicAxisCtrlPtr^.Input.Parameter.CyclicVel.SetVel);
			END_IF
			// Call Velocity Profiler
			fbSrampVelocityProfile();
			
			// Call Velocity Integrator
			fbVelocityIntegrator.fIn		:= fbSrampVelocityProfile.Y;
			fbVelocityIntegrator(stParams	:= VelocityIntegratorParams);
			
			// Copy Integrator Output to ExtSetPos
			{warning disable C0371}
			//Warning: Access to VAR_IN_OUT <Var> declared in <POU> from external context <Method/Transition/Property>
			AxisRef.PlcToNc.ExtSetDirection	:= 1;
			AxisRef.PlcToNc.ExtSetPos		:= fbVelocityIntegrator.fOut;
			{warning restore C0371}
			
	END_CASE
	
	// Call External Set Position function block
	{warning disable C0371}
	//Warning: Access to VAR_IN_OUT <Var> declared in <POU> from external context <Method/Transition/Property>
	fbMC_ExtSetPointGenEnable(Axis:= AxisRef); 
	{warning restore C0371}
	
	(* check if error occured *)
	IF IntErrorTrig_0.EDGEPOS(fbMC_ExtSetPointGenEnable.Error = TRUE) THEN
		// Add FB Error to ErrorHandler
		AddNCError(fbMC_ExtSetPointGenEnable.ErrorID, 'NC Error fbMC_ExtSetPointGenEnable ErrorID:');
		
		fbMC_ExtSetPointGenEnable.Execute	:= FALSE;
		CyclicVel	:= FALSE;
		AxisStep	:= CyclicAxis_STATE_ERROR;
	END_IF


	CyclicAxisCtrlPtr^.Output.Status.CyclicVel.Active	:= fbMC_ExtSetPointGenEnable.Enabled;
	CyclicAxisCtrlPtr^.Output.Status.CyclicVel.Busy		:= fbMC_ExtSetPointGenEnable.Busy;
END_METHOD

METHOD PRIVATE ResetAll_MC_FB : BOOL
VAR_INPUT
END_VAR

		ResetAll_MC_FB := FALSE ;
				
		fbMC_ExtSetPointGenEnable.Execute:= FALSE;
		fbMC_ExtSetPointGenDisable.Execute:= FALSE;
		{warning disable C0371}
		//Warning: Access to VAR_IN_OUT <Var> declared in <POU> from external context <Method/Transition/Property>
		fbMC_ExtSetPointGenEnable(Axis:= AxisRef); 
		fbMC_ExtSetPointGenDisable(Axis:= AxisRef) ;
		{warning restore C0371}
		
		
		memset(ADR(CyclicAxisCtrlPtr^.Input.Command) ,0 ,SIZEOF(CyclicAxisCtrlPtr^.Input.Command));
		memset(ADR(CyclicAxisCtrlPtr^.Output.Status) ,0 ,SIZEOF(CyclicAxisCtrlPtr^.Output.Status));
		
		ResetAll_MC_FB := TRUE ;
END_METHOD

END_FUNCTION_BLOCK

// ---- POUs/Lib/Motion/Engineering/SrampHp.TcPOU
FUNCTION_BLOCK SrampHp
VAR_INPUT
	X:			LREAL;
	A_UP:		LREAL;
	A_DN:		LREAL;
	VU_MAX:		LREAL;
	VD_MAX:		LREAL;
	LIMIT_HIGH:	LREAL;
	LIMIT_LOW:	LREAL;
	RST:		BOOL;
	SET:		BOOL;
END_VAR
VAR_OUTPUT
	Y:	LREAL;
	V:	LREAL;
END_VAR
VAR
	cycle_time: exTC_S;
	init: BOOL;
END_VAR

(* read the system_time in microseconds *)
cycle_time();

(* assure range of inputs *)
A_up := MAX(0.0, A_UP);
A_dn := MIN(0.0, A_dn);
VU_max := MAX(0.0, VU_max);
VD_max := MIN(0.0, VD_MAX);

(* calculate the output offset *)
IF SET THEN
	Y := X;
	V := 0.0;
ELSIF rst THEN
	
	Y := 0.0;
	V := 0.0;
ELSIF X = Y THEN
	v := 0.0;
ELSIF X > Y THEN
	(* output is too low >> ramp up and brake at the end *)
	(* accelerate the speed and limit to vu_max *)
	v := MIN(v + A_UP * cycle_time.TC, vu_max);
	(* calculate the max speed to be able to brake and select the lowest *)
	v := MIN(SQRT((Y-X) * 2.0 * A_DN), v);
	(* calculate the output and obey limits *)
	y := LIMIT(limit_low, y + MIN(v * cycle_time.TC, X-Y), limit_high);
ELSIF X < Y THEN
	(* output is too high >> ramp dn and brake at the end *)
	(* accelerate the speed and limit to vd_max *)
	v := MAX(v + A_DN * cycle_time.TC, vd_max);
	(* calculate the max speed to be able to brake and select the lowest *)
	v := MAX(-SQRT((Y-X) * 2.0 * A_UP), v);
	(* calculate the output and obey limits *)
	y := LIMIT(limit_low, y + MAX(v * cycle_time.TC, X-Y), limit_high);
END_IF;


(* revision history
hm	13. mar. 2008	rev 1.0
	original version

hm	11. mar. 2009	rev 1.1
	real constants updated to new systax using dot																																																																																																																																																																																																																																																																																																																																																																																																																																																																																																																																																																																																																																																																																																																																																																																																																																																																																																																																																																																																																																																											

*)

END_FUNCTION_BLOCK

// ---- POUs/Lib/Motion/External Libs/exTC_S.TcPOU
FUNCTION_BLOCK exTC_S
VAR_OUTPUT
	TC: REAL;
END_VAR
VAR
	init: BOOL;
	tx: DWORD;
	last: DWORD;
END_VAR

(* read system timer *)
tx := exT_PLC_US();

IF NOT init THEN
	init := TRUE;
	TC := 0.0;
ELSE
	tc := DWORD_TO_REAL(tx - last)*1.0E-6;
END_IF;
last := tx;

(* revision history
hm	13. mar. 2008	rev 1.0
	original version

hm	16. mar 2008	rev 1.1
	added type conversion to avoid warnings under codesys 3.0

hm	11. mar. 2009	rev 1.2
	changed real constants to use dot syntax

*)

END_FUNCTION_BLOCK

// ---- POUs/Lib/Motion/External Libs/exT_PLC_US.TcPOU
FUNCTION exT_PLC_US : DWORD
VAR CONSTANT
	debug: BOOL := 0;
	N: INT := 0;
	offset: DWORD := 0;
END_VAR
VAR
	tx: TIME;
END_VAR

tx := TIME();
exT_PLC_US := TIME_TO_DWORD(Tx)*1000;
(* hier muss die korrektur fr step7 stattfinden
plctime muss den vollen wertebereich von time ausnutzen:
wenn bei step7 time -24tage bis plus 24 tage ist dann muss der timer auch beim berlauf auf -24tage springen 
und auf keinen fall auf 0 !!!!
fr siemens muss ein weiterer fb im main eingebunden werden der sicherstellt das alle 32 bits durchgezהhlt werden.
es kann nur ein fb sein den er muss sich das oberste (32te) bit merken.
oder etwa spring s7 bei berlauf auf -24 tage????? dann wהre keine korrektur nצtig.
*)
IF debug THEN
	exT_PLC_US := (SHL(exT_PLC_US,N) OR SHL(DWORD#1,N)-1) + OFFSET;
END_IF;

(* revision history
hm	14.9.2007	rev 1.0
	original version

hm	12. nov 2007	rev 1.1
	added temporaray variable tx because some compilers could not handle time() as an argument

hm	16. nov. 2008	rev 1.2
	initialized constants with 0 for compatibility reasons

*)

END_FUNCTION

// ---- POUs/Lib/Motion/CanOpenAxis/Elmo/ElmoBasicAxis_FB.TcPOU
FUNCTION_BLOCK PUBLIC ElmoBasicAxis_FB EXTENDS CoE_BasicAxis_FB  
VAR_INPUT		
	pDigIn: 		    POINTER TO DINT;
	
END_VAR
VAR_IN_OUT	
END_VAR
VAR_OUTPUT	
END_VAR

VAR
	
	fbElmoIOsHandle:	FB_ElmoIOsHandle;
END_VAR


AxisCtrlPtr^.Input.Parameter.Drive.eDriveType := enumDriveType.eElmo;	
AxisCtrlPtr^.Input.Parameter.Drive.VendorNameID := eVendorNameID.Elmo;
SUPER^(AxisRef:=AxisRef);


IF pDigIn <> 0 THEN
	fbElmoIOsHandle(DigIn:=	pDigIn^);
	AxisCtrlPtr^.Output.Status.DriveEnable:=	fbElmoIOsHandle.bEnable;
END_IF

METHOD CreateDriveErrMsgDetails : enumMotorEvents
VAR_INPUT
	ErrorId			: UDINT;
END_VAR
CASE ErrorId OF
	16#0:
		CreateDriveErrMsgDetails := enumMotorEvents.NoEvents;
		
	16#2340:
		CreateDriveErrMsgDetails := enumMotorEvents.MotorSupplyError;
		fnLogMsg(ADR(LogMsg_0),LOG_ERROR,'Elmo Drive ErrorId %d  ,Short circuit',UDINT_TO_DINT(ErrorId),0,0);
	16#3120: 
		CreateDriveErrMsgDetails := enumMotorEvents.MotorSupplyError;
		fnLogMsg(ADR(LogMsg_0),LOG_ERROR,'Elmo Drive ErrorId %d Under Voltage',UDINT_TO_DINT(ErrorId),0,0);
	16#3130:
		CreateDriveErrMsgDetails := enumMotorEvents.MotorSupplyError;
		fnLogMsg(ADR(LogMsg_0),LOG_ERROR,'Elmo Drive ErrorId %d Hall  AC fail,loss off phase',UDINT_TO_DINT(ErrorId),0,0);
	16#3310:
		CreateDriveErrMsgDetails := enumMotorEvents.MotorOverCurrent ;
		fnLogMsg(ADR(LogMsg_0),LOG_ERROR,' voltage is too high',UDINT_TO_DINT(ErrorId),0,0);
 
	16#4310:
		CreateDriveErrMsgDetails := enumMotorEvents.MotorOverTemp ;
		fnLogMsg(ADR(LogMsg_0),LOG_ERROR,'Elmo Drive ErrorId %d Temp drive overhating',UDINT_TO_DINT(ErrorId),0,0);
	16#5280:
		CreateDriveErrMsgDetails := enumMotorEvents.MotorPositionError ;	
		fnLogMsg(ADR(LogMsg_0),LOG_ERROR,'Elmo Drive ErrorId %d Gantry position error',UDINT_TO_DINT(ErrorId),0,0);
		
	16#5441:
		CreateDriveErrMsgDetails := enumMotorEvents.DriveNotEnabled;
		fnLogMsg(ADR(LogMsg_0),LOG_ERROR,'Elmo Drive ErrorId %d Motor disables',UDINT_TO_DINT(ErrorId),0,0);
	16#5442:
		CreateDriveErrMsgDetails := enumMotorEvents.DriveNotEnabled;
		fnLogMsg(ADR(LogMsg_0),LOG_ERROR,'Elmo Drive ErrorId %d Motor disables by sw',UDINT_TO_DINT(ErrorId),0,0);
	16#6300:
		CreateDriveErrMsgDetails := enumMotorEvents.PLCIllegalParam;
		fnLogMsg(ADR(LogMsg_0),LOG_ERROR,'Elmo Drive ErrorId %d RPDO failed',UDINT_TO_DINT(ErrorId),0,0);
	16#7121:
		CreateDriveErrMsgDetails := enumMotorEvents.MotorPositionError;
		fnLogMsg(ADR(LogMsg_0),LOG_ERROR,'Elmo Drive ErrorId %d Motor stuck',UDINT_TO_DINT(ErrorId),0,0);
	16#7300:
		CreateDriveErrMsgDetails := enumMotorEvents.MotorFeedBackErr;
		fnLogMsg(ADR(LogMsg_0),LOG_ERROR,'Elmo Drive ErrorId %d Feedback error',UDINT_TO_DINT(ErrorId),0,0);
	16#7381:
 		CreateDriveErrMsgDetails := enumMotorEvents.DriveComError;
		fnLogMsg(ADR(LogMsg_0),LOG_ERROR,'Elmo Drive ErrorId %d 2 Dig halls sens where cng on the same time',UDINT_TO_DINT(ErrorId),0,0);
	16#7382: 
		CreateDriveErrMsgDetails := enumMotorEvents.MotorPositionError;
		fnLogMsg(ADR(LogMsg_0),LOG_ERROR,'Elmo Drive ErrorId %d Commutaition procees failed',UDINT_TO_DINT(ErrorId),0,0);
	16#8110:
		CreateDriveErrMsgDetails := enumMotorEvents.DriveComError;
		fnLogMsg(ADR(LogMsg_0),LOG_ERROR,'Elmo Drive ErrorId %d Cam Msg lost',UDINT_TO_DINT(ErrorId),0,0);
	16#8130:
		CreateDriveErrMsgDetails := enumMotorEvents.DriveComError;
		fnLogMsg(ADR(LogMsg_0),LOG_ERROR,'Elmo Drive ErrorId %d Heartbeat event',UDINT_TO_DINT(ErrorId),0,0);
	16#8140:
		CreateDriveErrMsgDetails := enumMotorEvents.MotorGeneralError;
		fnLogMsg(ADR(LogMsg_0),LOG_ERROR,'Elmo Drive ErrorId %d Recovered from bus off',UDINT_TO_DINT(ErrorId),0,0);
	16#8210:
		CreateDriveErrMsgDetails := enumMotorEvents.MotorGeneralError;
		fnLogMsg(ADR(LogMsg_0),LOG_ERROR,'Elmo Drive ErrorId %d access to non configured PDO',UDINT_TO_DINT(ErrorId),0,0);
	16#8311:
		CreateDriveErrMsgDetails := enumMotorEvents.MotorOverCurrent;
		fnLogMsg(ADR(LogMsg_0),LOG_ERROR,'Elmo Drive ErrorId %d Peak current has been exceeded',UDINT_TO_DINT(ErrorId),0,0);

	16#8480:
		CreateDriveErrMsgDetails := enumMotorEvents.MotorSpeedError;
		fnLogMsg(ADR(LogMsg_0),LOG_ERROR,'Elmo Drive ErrorId %d speed tracking Error',UDINT_TO_DINT(ErrorId),0,0);
	16#8481:
		CreateDriveErrMsgDetails := enumMotorEvents.MotorSpeedError;
		fnLogMsg(ADR(LogMsg_0),LOG_ERROR,'Elmo Drive ErrorId %d Speed limit Exceeded',UDINT_TO_DINT(ErrorId),0,0);
	16#8611:
		CreateDriveErrMsgDetails := enumMotorEvents.MotorPositionError;
		fnLogMsg(ADR(LogMsg_0),LOG_ERROR,'Elmo Drive ErrorId %d Position tracking error',UDINT_TO_DINT(ErrorId),0,0);
	16#8680:
		CreateDriveErrMsgDetails := enumMotorEvents.MotorPositionError;
		fnLogMsg(ADR(LogMsg_0),LOG_ERROR,'Elmo Drive ErrorId %d Position limit Exceeded',UDINT_TO_DINT(ErrorId),0,0);
	16#FF02:
		CreateDriveErrMsgDetails := enumMotorEvents.DriveComError;
		fnLogMsg(ADR(LogMsg_0),LOG_ERROR,'Elmo Drive ErrorId %d Com Error',UDINT_TO_DINT(ErrorId),0,0);
	16#FF10:
		CreateDriveErrMsgDetails := enumMotorEvents.MotorGeneralError ;
		fnLogMsg(ADR(LogMsg_0),LOG_ERROR,'Elmo Drive ErrorId %d Failed to start motor',UDINT_TO_DINT(ErrorId),0,0);
	16#FF20:
		CreateDriveErrMsgDetails := enumMotorEvents.MotorGeneralError;
		fnLogMsg(ADR(LogMsg_0),LOG_ERROR,'Elmo Drive ErrorId %d Saftey torque Off in use',UDINT_TO_DINT(ErrorId),0,0);
	16#FF40:
		CreateDriveErrMsgDetails := enumMotorEvents.MotorGeneralError;
		fnLogMsg(ADR(LogMsg_0),LOG_ERROR,'Elmo Drive ErrorId %d Gantry slave Disabled',UDINT_TO_DINT(ErrorId),0,0);
	ELSE
		fnLogMsg(ADR(LogMsg_0),LOG_ERROR,'unknown Elmo Drive ErrorId %d ',UDINT_TO_DINT(ErrorId),0,0);
		CreateDriveErrMsgDetails := enumMotorEvents.MotorGeneralError;
		 
END_CASE
END_METHOD

METHOD DriveUnitsTorqueToRealValue : LREAL
VAR_INPUT
	
	Torque: LREAL;	

END_VAR
DriveUnitsTorqueToRealValue := (Torque*AxisCtrlPtr^.Input.Parameter.RatedCurrent)/1000;
END_METHOD

METHOD GetCanOpenAdr : BOOL
VAR_INPUT
END_VAR


VAR
	
	SpeedSwSubIndex: INT;
END_VAR
    SUPER^.GetCanOpenAdr();	

	
	CoEDrive_Ctrl_Adr.KpSpeed.Index	   := 16#3113;	
	CoEDrive_Ctrl_Adr.KpSpeed.SunIndex  := 2;
	CoEDrive_Ctrl_Adr.KpSpeed.Size      := 4;
	CoEDrive_Ctrl_Adr.KpSpeed.IsReal    := TRUE;
	
	
	CoEDrive_Ctrl_Adr.KiSpeed.Index	    := 16#310C;	
	CoEDrive_Ctrl_Adr.KiSpeed.SunIndex  := 2;
   	CoEDrive_Ctrl_Adr.KiSpeed.Size      := 4;
	CoEDrive_Ctrl_Adr.KiSpeed.IsReal    := TRUE;
	
	CoEDrive_Ctrl_Adr.GainScheduler.Index	    := 16#30AE;	
	CoEDrive_Ctrl_Adr.GainScheduler.SunIndex    := 2;
   	CoEDrive_Ctrl_Adr.GainScheduler.Size        := 8;
	
	
	CoEDrive_Ctrl_Adr.AccClosePosErr.Index	    := 16#30AE;	
	CoEDrive_Ctrl_Adr.AccClosePosErr.SunIndex    := 9;
   	CoEDrive_Ctrl_Adr.AccClosePosErr.Size        := 8;
END_METHOD

METHOD GetErrCanAdr : BOOL
VAR_INPUT
END_VAR


VAR
	
END_VAR

	
	CoeErrIdIndex	 := 16#603F;
	CoeErrIdSubIndex := 0;
END_METHOD

METHOD  INIT_Specific : BOOL 
VAR_INPUT
	bStart: 					BOOL;
END_VAR
VAR_INST	
	ComDelay:	TON;
	Elmo_Init_State : INT ;
	ExecuteTrig: 	Trigger;
END_VAR
IF ExecuteTrig.EDGEPOS(bStart) THEN
	INIT_Specific := FALSE ;
	IF AxisCtrlPtr^.Input.Parameter.Drive.bDisableFoE_Transfer THEN 
		Elmo_Init_State:= 3;
	ELSE
		CoEDrive_Ctrl_Adr.ParamsVersionObj.Index    := 16#2F00;
		CoEDrive_Ctrl_Adr.ParamsVersionObj.SunIndex := 1; 		
		Elmo_Init_State:= 1;
	END_IF
END_IF


IF ExecuteTrig.EDGENEG(bStart) THEN
	Elmo_Init_State := 0;
END_IF	

	
CASE Elmo_Init_State OF							
	1:
		Meth_UpdateDriveParams(FALSE);
		Elmo_Init_State:=	2;
	2:	
		IF Meth_UpdateDriveParams(TRUE) THEN
			Elmo_Init_State:=	3;
		ELSIF AxisCtrlPtr^.Output.Status.Drive.eUpdate_Staus = enum_DriveUpdateStatus.Error THEN
			//
		END_IF

	3:
		ReadInitDriveParID(FALSE);
		Elmo_Init_State:=	4;
		
	4:
		IF ReadInitDriveParID(TRUE) THEN
			Elmo_Init_State:=	10;
		END_IF			

	10:
		
		Elmo_Init_State := 0 ;
		INIT_Specific := TRUE ;
		AxisCtrlPtr^.Output.Status.AxisInitDone := TRUE ;
		AxisCtrlPtr^.Output.Status.ReadyForCmd := TRUE ;
END_CASE
END_METHOD

METHOD Meth_ChangingOperationMode : BOOL
VAR_INPUT
	Execute   : BOOL;
	OperMode : eDriveModeOfOperation; 
	
END_VAR
VAR_INST
	
	ElmoCngOperState : INT;	
END_VAR

VAR
	
	ChangeDone : BOOL;
END_VAR
IF ChangeModeOperTrig.EDGEPOS(Execute) THEN

	Meth_ChangingOperationMode := FALSE;					
	ChangeDone := FALSE;
	ElmoCngOperState := 1;

	
END_IF


IF ChangeModeOperTrig.EDGENEG(Execute) THEN
	
	ElmoCngOperState := 0;
END_IF



CASE ElmoCngOperState OF
	0:
		Meth_CoEChangOperationMode(FALSE,eCaOpDriveModeOfOperation.ProfilePositionMode);
		
	1: 
		//Meth_CoEChangOperationMode
		CASE OperMode OF
			eDriveModeOfOperation.ProfilePositionMode				:
				IF Meth_CoEChangOperationMode(TRUE,eCaOpDriveModeOfOperation.ProfilePositionMode) THEN
					ChangeDone := TRUE;
				END_IF
				
		    eDriveModeOfOperation.VelocityCtrMode    				:
				IF Meth_CoEChangOperationMode(TRUE,eCaOpDriveModeOfOperation.ProfileVelocityMode)THEN
					ChangeDone := TRUE;
				END_IF
		    eDriveModeOfOperation.ProfileVelocityMode 	   	    :
				IF Meth_CoEChangOperationMode(TRUE,eCaOpDriveModeOfOperation.ProfileVelocityMode) THEN
					ChangeDone := TRUE;
				END_IF
				
		    eDriveModeOfOperation.TorqueVelocityMode 				:
				IF Meth_CoEChangOperationMode(TRUE,eCaOpDriveModeOfOperation.TorqueVelocityMode) THEN
					ChangeDone := TRUE;
				END_IF
				
		    eDriveModeOfOperation.HomingMode				    	:
				IF Meth_CoEChangOperationMode(TRUE,eCaOpDriveModeOfOperation.HomingMode)THEN
					ChangeDone := TRUE;
				END_IF
				
		    eDriveModeOfOperation.InterpolationPosMode			:
				IF Meth_CoEChangOperationMode(TRUE,eCaOpDriveModeOfOperation.InterpolationPosMode) THEN
					ChangeDone := TRUE;
				END_IF
		    eDriveModeOfOperation.CyclicSyncMode					:
				Meth_CoEChangOperationMode(TRUE,eCaOpDriveModeOfOperation.CyclicSyncMode);
		END_CASE
		ElmoCngOperState := 2;

	2:
 		Meth_ChangingOperationMode := TRUE;
		
		
END_CASE
END_METHOD

METHOD Meth_TorqueInDriveUnits : LREAL
VAR_INPUT
	
	Torque: LREAL;	

END_VAR
IF AxisCtrlPtr^.Input.Parameter.RatedCurrent <> 0 THEN
	Meth_TorqueInDriveUnits := (Torque*1000)/AxisCtrlPtr^.Input.Parameter.RatedCurrent;
END_IF
END_METHOD

METHOD ReadActualCurrent : LREAL
VAR_INPUT
END_VAR
VAR_INST
		
END_VAR


// Units [rms]

AxisCtrlPtr^.Output.monitor.ActualCurrent	:=  ( (THIS^.io_ActualCurrent) / 1000.0) * AxisCtrlPtr^.Input.Parameter.RatedCurrent / SQRT(2.0);
END_METHOD

METHOD ReadActualTorque : LREAL
VAR_INPUT
END_VAR
VAR_INST
		
END_VAR

// Units [rms]
//AxisCtrlPtr^.Output.monitor.ActualCurrent Get from ReadActualCurrent method
// on Elmo it is needed to link only IO  io_ActualCurrent
AxisCtrlPtr^.Output.monitor.ActualTorque	:=  AxisCtrlPtr^.Output.monitor.ActualCurrent * AxisCtrlPtr^.Input.Parameter.Drive.Kt;
END_METHOD

METHOD ReadInitDriveParID : BOOL
VAR_INPUT
	bStart : BOOL;
END_VAR

VAR_INST
	ExecuteTrig_1: 		Trigger;
	State_InitSpecific_1: INT;
END_VAR

IF ExecuteTrig_1.EDGEPOS(bStart) THEN
	ReadInitDriveParID		:= FALSE;
	State_InitSpecific_1	:= 1;		
END_IF

IF ExecuteTrig_1.EDGENEG(bStart) THEN
	State_InitSpecific_1	:= 0;	
	ReadInitDriveParID		:= FALSE;
END_IF

CASE State_InitSpecific_1 OF

	 
	
	1:
		SUPER^.EcCoeSdoRead(FALSE);
		CoeSdoRW.Input.Read.nIndex		:= DINT_TO_WORD(eElmoDriveParID.RatedCurrent);
		CoeSdoRW.Input.Read.nSubIndex	:= 0;
		CoeSdoRW.Input.Read.pDstBuf		:= ADR(CoeRead_RatedCurrent);
		CoeSdoRW.Input.Read.cbBufLen	:= SIZEOF(CoeRead_RatedCurrent);
		State_InitSpecific_1	:= 2;
		
	2:
		IF SUPER^.EcCoeSdoRead(TRUE) THEN	
			State_InitSpecific_1	:= 3;
		END_IF
		
	3:
		SUPER^.EcCoeSdoRead(FALSE);
		CoeSdoRW.Input.Read.nIndex		:= DINT_TO_WORD(eElmoDriveParID.RatedTorque);
		CoeSdoRW.Input.Read.nSubIndex	:= 0;
		CoeSdoRW.Input.Read.pDstBuf		:= ADR(CoeRead_RatedTorque);
		CoeSdoRW.Input.Read.cbBufLen	:= SIZEOF(CoeRead_RatedTorque);
		State_InitSpecific_1	:= 4;
		
	4:
		IF SUPER^.EcCoeSdoRead(TRUE) THEN
			AxisCtrlPtr^.Input.Parameter.RatedCurrent	:= UDINT_TO_LREAL(CoeRead_RatedCurrent) / 1000.0;
			AxisCtrlPtr^.Input.Parameter.Ratedtorque	:= UDINT_TO_LREAL(CoeRead_RatedTorque) / 1000.0;
			ReadInitDriveParID		:= TRUE;	
			State_InitSpecific_1	:= 0;
		END_IF
		
END_CASE
END_METHOD

END_FUNCTION_BLOCK

// ---- POUs/Lib/Motion/CanOpenAxis/CoE_BasicAxis_FB.TcPOU
FUNCTION_BLOCK PUBLIC CoE_BasicAxis_FB EXTENDS BasicAxis_FB  
VAR_INPUT
	io_StatusWord : UINT;	
END_VAR
VAR_IN_OUT
	
END_VAR

VAR_OUTPUT	
	OperationMode : USINT :=8;
END_VAR

VAR
	CoeErrIdIndex		: WORD;
	CoeErrIdSubIndex	: BYTE;
		
	CoeRead_RatedTorque			: UDINT;
	CoeRead_RatedCurrent		: UDINT;					
	UsintValue					: USINT;// For read write sdo
	UdintValue					: UDINT;// For read write sdo
	UintValue					: UINT;// For read write sdo
	Ulong						: ULINT;
	LRealValue					: LREAL;// For read write sdo
	RealValue					: REAL;// For read write sdo
	ReadObjError                : BOOL;
	FB_EcCoeSdoWrite			: FB_EcCoESdoWrite;
	//
	CoEDrive_Ctrl_Adr:    CoEDrive_Ctrl_Adr_typ;
	
	Homing_Ctrl_Params: Homing_CoE_Ctrl_Paramters_typ;
	
	NextState    : INT;
	ErrorOnState : INT;
	InitCanOpenAdr: BOOL := FALSE;
 
	//FOE
	FOE_Ctrl_Paramters: CoE_FOE_Ctrl_typ;		
	FOE_Ctrl_UpdateFW:  CoE_FOE_Ctrl_typ;
	
	 LogText		: STRING(500);
END_VAR



IF InitCanOpenAdr = FALSE THEN
	GetCanOpenAdr();
	InitCanOpenAdr := TRUE;
END_IF

SUPER^(AxisRef:=AxisRef);
FB_EcCoeSdoWrite();	// For Meth_ChangingOperationMode. Need to change to EcCoeSdoWrite !!! 
ReadActualTorque() ;
ReadActualCurrent() ;
//FOE
Meth_FOE_fbCalls();

METHOD CreateDriveErrMsgDetails : enumMotorEvents
VAR_INPUT
	ErrorId			: UDINT;
END_VAR
fnLogMsg(ADR(LogMsg_0),LOG_ERROR,'ErrorId %d  ',UDINT_TO_DINT(ErrorId),0,0);
//Etz to do
CreateDriveErrMsgDetails := enumMotorEvents.NoEvents;
END_METHOD

METHOD DriveErrorHandling : BOOL

VAR_INST
	ErrHandState	: INT;
	
	FB_SoEReset_0	: FB_SoEReset;
	FB_EcSoERead_DriveError		: FB_EcSoERead;
	tmpDriveErrorId				: UDINT;
	LastError       			: UDINT; 
	LastErrorCounter            : UDINT := 0; 
	FB_EcCoeSdoRead_DriveError	: FB_EcCoeSdoRead;
	MC_Reset_0					: MC_Reset;
	tmpErrorEntry			: Eh_ErrorEntry_typ;
END_VAR


CASE ErrHandState OF
	0: // logic init
		GetErrCanAdr();	
		ErrHandState	:= 200;
		
		
	//************************* CAN Logic **********************************************
	200: // wait errors
		{warning disable C0371}
		IF AxisRef.Status.DriveDeviceError THEN
			(*IF AxisCtrlPtr^.Output.Status.Drive.ActiveHW AND io_HW_State <> 8 THEN
				 tmp_ErrorEntry.ErrorText	:= AxisCtrlPtr^.Input.Parameter.ThreadName;
				 tmp_ErrorEntry.ErrorText	:= CONCAT(tmp_ErrorEntry.ErrorText,'Drive Not In OP ');
				 tmp_ErrorEntry.MotorEvents  :=enumMotorEvents.DriveComError ;
				 fnLogMsg(ADR(LogMsg_0),LOG_ERROR,tmp_ErrorEntry.ErrorText,0,0,0);
				 		
				 AxisCtrlPtr^.Output.Error.fbErrorHandler.ErrorPush(tmp_ErrorEntry);	
				
				 ErrHandState	:= 205;
			ELSE*)
				FB_SoEReset_0.Execute				:= FALSE;
				FB_EcSoERead_DriveError.bExecute	:= FALSE;
				ErrHandState	:= 210;
	
		//	END_IF	
		
		ELSIF AxisRef.NcToPlc.ErrorCode <> 0 
			AND AxisRef.NcToPlc.ErrorCode <> 18000 THEN
			// ETZ Axis.NcToPlc.ErrorCode
			ErrHandState	:= 300;
		ELSIF AxisCtrlPtr^.Output.Error.fbErrorHandler.EntriesCount > 0 THEN
			// do nothing
		END_IF
	
		IF AxisRef.Status.DriveDeviceError = FALSE THEN
			LastError := 0;
			LastErrorCounter := 0;
		END_IF
		{warning restore C0371}
	205: // Wait for OP
		IF io_HW_State = 8 THEN
			ErrHandState	:= 200;
		END_IF
	210: // wait speed decrease
		IF AxisCtrlPtr^.Output.monitor.ActVelocity < 500 THEN
			ErrHandState	:= 211;	// read can error
		END_IF
		
	211:// read error according to drive Error Index
		
		// Fix link problem
		IF strEcNetId= '' AND (AxisCtrlPtr^.Input.Parameter.ecNetIdArr[4]<>0 OR AxisCtrlPtr^.Input.Parameter.ecNetIdArr[5]<>0) THEN
			strEcNetId:= F_CreateAmsNetId(AxisCtrlPtr^.Input.Parameter.ecNetIdArr);
		END_IF	

		FB_EcCoeSdoRead_DriveError.sNetId		:= strEcNetId;
		FB_EcCoeSdoRead_DriveError.nSlaveAddr	:= AxisCtrlPtr^.Input.Parameter.Drive.EtherCatAddr;
		FB_EcCoeSdoRead_DriveError.nIndex		:= CoeErrIdIndex; 
		FB_EcCoeSdoRead_DriveError.nSubIndex	:= CoeErrIdSubIndex; 
		FB_EcCoeSdoRead_DriveError.pDstBuf		:= ADR(tmpDriveErrorId);
		FB_EcCoeSdoRead_DriveError.cbBufLen		:= SIZEOF(tmpDriveErrorId);
		FB_EcCoeSdoRead_DriveError.tTimeout		:= T#10S;
		
		FB_EcCoeSdoRead_DriveError.bExecute		:= TRUE;
		
		ErrHandState	:= 212;
	212:
		IF NOT FB_EcCoeSdoRead_DriveError.bBusy THEN
			FB_EcCoeSdoRead_DriveError.bExecute		:= FALSE;
			IF NOT FB_EcCoeSdoRead_DriveError.bError THEN
				// Add Drive Error to ErrorHandler
				tmp_ErrorEntry.ErrorId		:= tmpDriveErrorId;
			//	IF LastError <>  tmp_ErrorEntry.ErrorId OR LastErrorCounter > 100 THEN
					tmp_ErrorEntry.ErrorText	:= AxisCtrlPtr^.Input.Parameter.ThreadName;
					tmp_ErrorEntry.ErrorText	:= CONCAT(tmp_ErrorEntry.ErrorText,' Drive ErrorID: ');
					tmp_ErrorEntry.ErrorText	:= CONCAT(tmp_ErrorEntry.ErrorText, UDINT_TO_STRING(tmp_ErrorEntry.ErrorId));
					tmp_ErrorEntry.ErrorText	:= CONCAT(tmp_ErrorEntry.ErrorText, ', Or 0x');
					tmp_ErrorEntry.ErrorText	:= CONCAT(tmp_ErrorEntry.ErrorText, UDINT_TO_HEX_STRING(tmp_ErrorEntry.ErrorId));
					
					tmp_ErrorEntry.MotorEvents  := CreateDriveErrMsgDetails(tmp_ErrorEntry.ErrorId);
					fnLogMsg(ADR(LogMsg_0),LOG_ERROR,tmp_ErrorEntry.ErrorText,0,0,0);
					//ETZ to Add method for Log			
					AxisCtrlPtr^.Output.Error.fbErrorHandler.ErrorPush(tmp_ErrorEntry);
					LastError :=  tmp_ErrorEntry.ErrorId;
					LastErrorCounter := 0;
			(*	ELSE
					LastErrorCounter := LastErrorCounter + 1;	
				END_IF*)
				
		
			ELSE // IF bError
				fnLogMsg(ADR(LogMsg_0),LOG_ERROR,'NO LINKS FOR DRIVE',0,0,0);				 
			END_IF
			ErrHandState	:= 300;	// MC_Reset
		END_IF
 
	300: // Run MC_Reset
		MC_Reset_0.Execute	:= TRUE;
		ErrHandState		:= 301;
	301:
		{warning disable C0371}
		IF MC_Reset_0.Done 
			AND AxisRef.NcToPlc.ErrorCode = 0
			(*AND Axis.Status.DriveDeviceError = FALSE*) THEN
			MC_Reset_0.Execute	:= FALSE;
	
			ErrHandState	:= 0;
		
		ELSIF MC_Reset_0.Error THEN
			MC_Reset_0.Execute	:= FALSE;
			// Add FB Error to ErrorHandler
			tmp_ErrorEntry.ErrorId		:= MC_Reset_0.ErrorID;
			tmp_ErrorEntry.ErrorText	:= 'FB MC_Reset_0 ErrorID: ';
			tmp_ErrorEntry.ErrorText	:= CONCAT(tmp_ErrorEntry.ErrorText, UDINT_TO_STRING(tmp_ErrorEntry.ErrorId));
			AxisCtrlPtr^.Output.Error.fbErrorHandler.ErrorPush(tmp_ErrorEntry);
			
			ErrHandState	:= 0;
		END_IF
		{warning restore C0371}
		
		IF (AxisCtrlPtr^.Output.Status.CommunicationError = TRUE) THEN
			MC_Reset_0.Execute	:= FALSE;
			ErrHandState		:= 400;	
		END_IF
		
		IF NOT AxisCtrlPtr^.Output.Status.DriveEnable THEN
			MC_Reset_0.Execute	:= FALSE;
			ErrHandState		:= 500;	
		END_IF
	400:
		IF (AxisCtrlPtr^.Output.Status.CommunicationError = FALSE) THEN
			ErrHandState	:= 300;	
		END_IF
	500:
		IF AxisCtrlPtr^.Output.Status.DriveEnable THEN
			MC_Reset_0.Execute	:= FALSE;
			ErrHandState		:= 200;	
		END_IF
	
END_CASE

FB_EcSoERead_DriveError();
FB_EcCoeSdoRead_DriveError();
{warning disable C0371}
FB_SoEReset_0(Axis:= AxisRef);
MC_Reset_0(Axis:= AxisRef);
{warning restore C0371}
END_METHOD

